gfCNCPoint1[10884] = {X 272.2327, Y 98.0000, Z -1.3333, A 0.000, B 0.000, C 0.000 }
gfCNCPoint1[10885] = {X 272.2329, Y 97.0232, Z -1.3333, A 0.000, B 0.000, C 0.000 }
gfCNCPoint1[10886] = {X 272.3321, Y 96.1797, Z -1.3333, A 0.000, B 0.000, C 0.000 }
gfCNCPoint1[10887] = {X 272.6072, Y 95.3761, Z -1.3333, A 0.000, B 0.000, C 0.000 }
gfCNCPoint1[10888] = {X 273.0457, Y 94.6486, Z -1.3333, A 0.000, B 0.000, C 0.000 }
gfCNCPoint1[10889] = {X 273.6280, Y 94.0302, Z -1.3333, A 0.000, B 0.000, C 0.000 }
gfCNCPoint1[10890] = {X 274.3277, Y 93.5487, Z -1.3333, A 0.000, B 0.000, C 0.000 }
gfCNCPoint1[10891] = {X 275.1133, Y 93.2258, Z -1.3333, A 0.000, B 0.000, C 0.000 }
gfCNCPoint1[10892] = {X 275.9494, Y 93.0760, Z -1.3333, A 0.000, B 0.000, C 0.000 }
gfCNCPoint1[10893] = {X 275.9494, Y 85.3767, Z -1.3333, A 0.000, B 0.000, C 0.000 }
gfCNCPoint1[10894] = {X 262.6059, Y 80.1460, Z -1.3333, A 0.000, B 0.000, C 0.000 }
gfCNCPoint1[10895] = {X 262.1034, Y 80.4620, Z -1.3333, A 0.000, B 0.000, C 0.000 }
gfCNCPoint1[10896] = {X 237.4742, Y 96.4149, Z -1.3333, A 0.000, B 0.000, C 0.000 }
gfCNCPoint1[10897] = {X 237.4798, Y 97.0659, Z -1.3333, A 0.000, B 0.000, C 0.000 }
gfCNCPoint1[10898] = {X 237.4798, Y 98.0000, Z -1.3333, A 0.000, B 0.000, C 0.000 }
gfCNCPoint1[10899] = {X 237.3795, Y 98.8901, Z -1.3333, A 0.000, B 0.000, C 0.000 }
gfCNCPoint1[10900] = {X 237.0837, Y 99.7355, Z -1.3333, A 0.000, B 0.000, C 0.000 }
gfCNCPoint1[10901] = {X 236.6071, Y 100.4940, Z -1.3333, A 0.000, B 0.000, C 0.000 }
gfCNCPoint1[10902] = {X 235.9737, Y 101.1273, Z -1.3333, A 0.000, B 0.000, C 0.000 }
gfCNCPoint1[10903] = {X 235.2153, Y 101.6039, Z -1.3333, A 0.000, B 0.000, C 0.000 }
gfCNCPoint1[10904] = {X 234.3699, Y 101.8997, Z -1.3333, A 0.000, B 0.000, C 0.000 }
gfCNCPoint1[10905] = {X 233.4798, Y 102.0000, Z -1.3333, A 0.000, B 0.000, C 0.000 }
gfCNCPoint1[10906] = {X 214.1790, Y 102.0000, Z -1.3333, A 0.000, B 0.000, C 0.000 }
gfCNCPoint1[10907] = {X 213.7859, Y 101.9806, Z -1.3333, A 0.000, B 0.000, C 0.000 }
gfCNCPoint1[10908] = {X 213.3966, Y 101.9227, Z -1.3333, A 0.000, B 0.000, C 0.000 }
gfCNCPoint1[10909] = {X 213.0072, Y 101.9806, Z -1.3333, A 0.000, B 0.000, C 0.000 }
gfCNCPoint1[10910] = {X 212.6141, Y 102.0000, Z -1.3333, A 0.000, B 0.000, C 0.000 }
gfCNCPoint1[10911] = {X 194.9870, Y 102.0000, Z -1.3333, A 0.000, B 0.000, C 0.000 }
gfCNCPoint1[10912] = {X 194.0969, Y 101.8997, Z -1.3333, A 0.000, B 0.000, C 0.000 }
gfCNCPoint1[10913] = {X 193.2514, Y 101.6039, Z -1.3333, A 0.000, B 0.000, C 0.000 }
gfCNCPoint1[10914] = {X 192.4930, Y 101.1273, Z -1.3333, A 0.000, B 0.000, C 0.000 }
gfCNCPoint1[10915] = {X 191.8596, Y 100.4940, Z -1.3333, A 0.000, B 0.000, C 0.000 }
gfCNCPoint1[10916] = {X 191.3831, Y 99.7355, Z -1.3333, A 0.000, B 0.000, C 0.000 }
gfCNCPoint1[10917] = {X 191.0872, Y 98.8901, Z -1.3333, A 0.000, B 0.000, C 0.000 }
gfCNCPoint1[10918] = {X 190.9870, Y 98.0000, Z -1.3333, A 0.000, B 0.000, C 0.000 }
gfCNCPoint1[10919] = {X 190.9870, Y 97.0659, Z -1.3333, A 0.000, B 0.000, C 0.000 }
gfCNCPoint1[10920] = {X 191.0804, Y 96.2066, Z -1.3333, A 0.000, B 0.000, C 0.000 }
gfCNCPoint1[10921] = {X 191.3562, Y 95.3874, Z -1.3333, A 0.000, B 0.000, C 0.000 }
gfCNCPoint1[10922] = {X 191.8015, Y 94.6466, Z -1.3333, A 0.000, B 0.000, C 0.000 }
gfCNCPoint1[10923] = {X 191.8852, Y 94.5402, Z -1.3333, A 0.000, B 0.000, C 0.000 }
gfCNCPoint1[10924] = {X 191.9725, Y 94.4367, Z -1.3333, A 0.000, B 0.000, C 0.000 }
gfCNCPoint1[10925] = {X 192.0154, Y 94.3938, Z -1.3333, A 0.000, B 0.000, C 0.000 }
gfCNCPoint1[10926] = {X 188.7055, Y 90.7802, Z -1.3333, A 0.000, B 0.000, C 0.000 }
gfCNCPoint1[10927] = {X 149.9476, Y 90.7802, Z -1.3333, A 0.000, B 0.000, C 0.000 }
gfCNCPoint1[10928] = {X 146.7183, Y 94.3579, Z -1.3333, A 0.000, B 0.000, C 0.000 }
gfCNCPoint1[10929] = {X 147.1679, Y 94.9493, Z -1.3333, A 0.000, B 0.000, C 0.000 }
gfCNCPoint1[10930] = {X 147.5014, Y 95.6130, Z -1.3333, A 0.000, B 0.000, C 0.000 }
gfCNCPoint1[10931] = {X 147.7075, Y 96.3267, Z -1.3333, A 0.000, B 0.000, C 0.000 }
gfCNCPoint1[10932] = {X 147.7791, Y 97.0661, Z -1.3333, A 0.000, B 0.000, C 0.000 }
gfCNCPoint1[10933] = {X 147.7791, Y 98.0000, Z -1.3333, A 0.000, B 0.000, C 0.000 }
gfCNCPoint1[10934] = {X 147.6788, Y 98.8901, Z -1.3333, A 0.000, B 0.000, C 0.000 }
gfCNCPoint1[10935] = {X 147.3830, Y 99.7355, Z -1.3333, A 0.000, B 0.000, C 0.000 }
gfCNCPoint1[10936] = {X 146.9064, Y 100.4940, Z -1.3333, A 0.000, B 0.000, C 0.000 }
gfCNCPoint1[10937] = {X 146.2731, Y 101.1273, Z -1.3333, A 0.000, B 0.000, C 0.000 }
gfCNCPoint1[10938] = {X 145.5146, Y 101.6039, Z -1.3333, A 0.000, B 0.000, C 0.000 }
gfCNCPoint1[10939] = {X 144.6692, Y 101.8997, Z -1.3333, A 0.000, B 0.000, C 0.000 }
gfCNCPoint1[10940] = {X 143.7791, Y 102.0000, Z -1.3333, A 0.000, B 0.000, C 0.000 }
gfCNCPoint1[10941] = {X 125.0000, Y 102.0000, Z -1.3333, A 0.000, B 0.000, C 0.000 }
gfCNCPoint1[10942] = {X 124.1099, Y 101.8997, Z -1.3333, A 0.000, B 0.000, C 0.000 }
gfCNCPoint1[10943] = {X 123.2645, Y 101.6039, Z -1.3333, A 0.000, B 0.000, C 0.000 }
gfCNCPoint1[10944] = {X 122.5060, Y 101.1273, Z -1.3333, A 0.000, B 0.000, C 0.000 }
gfCNCPoint1[10945] = {X 121.8727, Y 100.4940, Z -1.3333, A 0.000, B 0.000, C 0.000 }
gfCNCPoint1[10946] = {X 121.3961, Y 99.7355, Z -1.3333, A 0.000, B 0.000, C 0.000 }
gfCNCPoint1[10947] = {X 121.1003, Y 98.8901, Z -1.3333, A 0.000, B 0.000, C 0.000 }
gfCNCPoint1[10948] = {X 121.0000, Y 98.0000, Z -1.3333, A 0.000, B 0.000, C 0.000 }
gfCNCPoint1[10949] = {X 121.0000, Y 97.0659, Z -1.3333, A 0.000, B 0.000, C 0.000 }
gfCNCPoint1[10950] = {X 121.0981, Y 96.1853, Z -1.3333, A 0.000, B 0.000, C 0.000 }
gfCNCPoint1[10951] = {X 121.3877, Y 95.3479, Z -1.3333, A 0.000, B 0.000, C 0.000 }
gfCNCPoint1[10952] = {X 121.8546, Y 94.5948, Z -1.3333, A 0.000, B 0.000, C 0.000 }
gfCNCPoint1[10953] = {X 122.4758, Y 93.9629, Z -1.3333, A 0.000, B 0.000, C 0.000 }
gfCNCPoint1[10954] = {X 123.2209, Y 93.4834, Z -1.3333, A 0.000, B 0.000, C 0.000 }
gfCNCPoint1[10955] = {X 124.0533, Y 93.1796, Z -1.3333, A 0.000, B 0.000, C 0.000 }
gfCNCPoint1[10956] = {X 124.9321, Y 93.0665, Z -1.3333, A 0.000, B 0.000, C 0.000 }
gfCNCPoint1[10957] = {X 124.9750, Y 93.0393, Z -1.3333, A 0.000, B 0.000, C 0.000 }
gfCNCPoint1[10958] = {X 125.4940, Y 92.9623, Z -1.3333, A 0.000, B 0.000, C 0.000 }
gfCNCPoint1[10959] = {X 126.3825, Y 92.8105, Z -1.3333, A 0.000, B 0.000, C 0.000 }
gfCNCPoint1[10960] = {X 127.2582, Y 92.5973, Z -1.3333, A 0.000, B 0.000, C 0.000 }
gfCNCPoint1[10961] = {X 128.5219, Y 91.4099, Z -1.3333, A 0.000, B 0.000, C 0.000 }
gfCNCPoint1[10962] = {X 129.7180, Y 90.1544, Z -1.3333, A 0.000, B 0.000, C 0.000 }
gfCNCPoint1[10963] = {X 133.8038, Y 85.6598, Z -1.3333, A 0.000, B 0.000, C 0.000 }
gfCNCPoint1[10964] = {X 140.9145, Y 77.8539, Z -1.3333, A 0.000, B 0.000, C 0.000 }
gfCNCPoint1[10965] = {X 137.8983, Y 75.1063, Z -1.3333, A 0.000, B 0.000, C 0.000 }
gfCNCPoint1[10966] = {X 137.8983, Y 75.1063, Z 1.6667, A 0.000, B 0.000, C 0.000 }
gfCNCPoint1[10967] = {X 137.8983, Y 75.1063, Z 11.0000, A 0.000, B 0.000, C 0.000 }
gfCNCPoint1[10968] = {X 167.3809, Y 20.2812, Z 11.0000, A 0.000, B 0.000, C 0.000 }
gfCNCPoint1[10969] = {X 167.3809, Y 20.2812, Z 1.6667, A 0.000, B 0.000, C 0.000 }
gfCNCPoint1[10970] = {X 167.3809, Y 20.2812, Z -1.3333, A 0.000, B 0.000, C 0.000 }
gfCNCPoint1[10971] = {X 171.1581, Y 18.7388, Z -1.3333, A 0.000, B 0.000, C 0.000 }
gfCNCPoint1[10972] = {X 169.8405, Y 15.5121, Z -1.3333, A 0.000, B 0.000, C 0.000 }
gfCNCPoint1[10973] = {X 169.5912, Y 14.6607, Z -1.3333, A 0.000, B 0.000, C 0.000 }
gfCNCPoint1[10974] = {X 169.5212, Y 13.7764, Z -1.3333, A 0.000, B 0.000, C 0.000 }
gfCNCPoint1[10975] = {X 169.6332, Y 12.8964, Z -1.3333, A 0.000, B 0.000, C 0.000 }
gfCNCPoint1[10976] = {X 169.9226, Y 12.0578, Z -1.3333, A 0.000, B 0.000, C 0.000 }
gfCNCPoint1[10977] = {X 170.3773, Y 11.2960, Z -1.3333, A 0.000, B 0.000, C 0.000 }
gfCNCPoint1[10978] = {X 170.9779, Y 10.6432, Z -1.3333, A 0.000, B 0.000, C 0.000 }
gfCNCPoint1[10979] = {X 171.6992, Y 10.1268, Z -1.3333, A 0.000, B 0.000, C 0.000 }
gfCNCPoint1[10980] = {X 172.3295, Y 9.7674, Z -1.3333, A 0.000, B 0.000, C 0.000 }
gfCNCPoint1[10981] = {X 173.2114, Y 9.3960, Z -1.3333, A 0.000, B 0.000, C 0.000 }
gfCNCPoint1[10982] = {X 174.1534, Y 9.2278, Z -1.3333, A 0.000, B 0.000, C 0.000 }
gfCNCPoint1[10983] = {X 175.1093, Y 9.2711, Z -1.3333, A 0.000, B 0.000, C 0.000 }
gfCNCPoint1[10984] = {X 176.0323, Y 9.5238, Z -1.3333, A 0.000, B 0.000, C 0.000 }
gfCNCPoint1[10985] = {X 178.2250, Y 8.6014, Z -1.3333, A 0.000, B 0.000, C 0.000 }
gfCNCPoint1[10986] = {X 180.4990, Y 7.9029, Z -1.3333, A 0.000, B 0.000, C 0.000 }
gfCNCPoint1[10987] = {X 182.8314, Y 7.4353, Z -1.3333, A 0.000, B 0.000, C 0.000 }
gfCNCPoint1[10988] = {X 185.1988, Y 7.2031, Z -1.3333, A 0.000, B 0.000, C 0.000 }
gfCNCPoint1[10989] = {X 187.5777, Y 7.2088, Z -1.3333, A 0.000, B 0.000, C 0.000 }
gfCNCPoint1[10990] = {X 189.9440, Y 7.4523, Z -1.3333, A 0.000, B 0.000, C 0.000 }
gfCNCPoint1[10991] = {X 191.7010, Y 7.8143, Z -1.3333, A 0.000, B 0.000, C 0.000 }
gfCNCPoint1[10992] = {X 193.4116, Y 8.3544, Z -1.3333, A 0.000, B 0.000, C 0.000 }
gfCNCPoint1[10993] = {X 195.0579, Y 9.0671, Z -1.3333, A 0.000, B 0.000, C 0.000 }
gfCNCPoint1[10994] = {X 196.6223, Y 9.9449, Z -1.3333, A 0.000, B 0.000, C 0.000 }
gfCNCPoint1[10995] = {X 198.0886, Y 10.9785, Z -1.3333, A 0.000, B 0.000, C 0.000 }
gfCNCPoint1[10996] = {X 199.1482, Y 11.9218, Z -1.3333, A 0.000, B 0.000, C 0.000 }
gfCNCPoint1[10997] = {X 200.0991, Y 12.9747, Z -1.3333, A 0.000, B 0.000, C 0.000 }
gfCNCPoint1[10998] = {X 200.9301, Y 14.1245, Z -1.3333, A 0.000, B 0.000, C 0.000 }
gfCNCPoint1[10999] = {X 201.6314, Y 15.3578, Z -1.3333, A 0.000, B 0.000, C 0.000 }
gfCNCPoint1[11000] = {X 202.1947, Y 16.6598, Z -1.3333, A 0.000, B 0.000, C 0.000 }
gfCNCPoint1[11001] = {X 202.6689, Y 18.3162, Z -1.3333, A 0.000, B 0.000, C 0.000 }
gfCNCPoint1[11002] = {X 202.9504, Y 20.0160, Z -1.3333, A 0.000, B 0.000, C 0.000 }
gfCNCPoint1[11003] = {X 203.0354, Y 21.7368, Z -1.3333, A 0.000, B 0.000, C 0.000 }
gfCNCPoint1[11004] = {X 202.9228, Y 23.4560, Z -1.3333, A 0.000, B 0.000, C 0.000 }
gfCNCPoint1[11005] = {X 202.6141, Y 25.1511, Z -1.3333, A 0.000, B 0.000, C 0.000 }
gfCNCPoint1[11006] = {X 202.1724, Y 26.5972, Z -1.3333, A 0.000, B 0.000, C 0.000 }
gfCNCPoint1[11007] = {X 201.5477, Y 27.9741, Z -1.3333, A 0.000, B 0.000, C 0.000 }
gfCNCPoint1[11008] = {X 200.7505, Y 29.2589, Z -1.3333, A 0.000, B 0.000, C 0.000 }
gfCNCPoint1[11009] = {X 199.7941, Y 30.4301, Z -1.3333, A 0.000, B 0.000, C 0.000 }
gfCNCPoint1[11010] = {X 198.6946, Y 31.4680, Z -1.3333, A 0.000, B 0.000, C 0.000 }
gfCNCPoint1[11011] = {X 199.4963, Y 31.8092, Z -1.3333, A 0.000, B 0.000, C 0.000 }
gfCNCPoint1[11012] = {X 200.2132, Y 32.3043, Z -1.3333, A 0.000, B 0.000, C 0.000 }
gfCNCPoint1[11013] = {X 200.8162, Y 32.9331, Z -1.3333, A 0.000, B 0.000, C 0.000 }
gfCNCPoint1[11014] = {X 201.2808, Y 33.6702, Z -1.3333, A 0.000, B 0.000, C 0.000 }
gfCNCPoint1[11015] = {X 204.3222, Y 39.9530, Z -1.3333, A 0.000, B 0.000, C 0.000 }
gfCNCPoint1[11016] = {X 204.6427, Y 40.8622, Z -1.3333, A 0.000, B 0.000, C 0.000 }
gfCNCPoint1[11017] = {X 204.7537, Y 41.8197, Z -1.3333, A 0.000, B 0.000, C 0.000 }
gfCNCPoint1[11018] = {X 204.6496, Y 42.7781, Z -1.3333, A 0.000, B 0.000, C 0.000 }
gfCNCPoint1[11019] = {X 204.3355, Y 43.6895, Z -1.3333, A 0.000, B 0.000, C 0.000 }
gfCNCPoint1[11020] = {X 203.8272, Y 44.5085, Z -1.3333, A 0.000, B 0.000, C 0.000 }
gfCNCPoint1[11021] = {X 203.1499, Y 45.1945, Z -1.3333, A 0.000, B 0.000, C 0.000 }
gfCNCPoint1[11022] = {X 202.6134, Y 45.6282, Z -1.3333, A 0.000, B 0.000, C 0.000 }
gfCNCPoint1[11023] = {X 201.9086, Y 46.0913, Z -1.3333, A 0.000, B 0.000, C 0.000 }
gfCNCPoint1[11024] = {X 201.1276, Y 46.4092, Z -1.3333, A 0.000, B 0.000, C 0.000 }
gfCNCPoint1[11025] = {X 200.2998, Y 46.5700, Z -1.3333, A 0.000, B 0.000, C 0.000 }
gfCNCPoint1[11026] = {X 199.4565, Y 46.5675, Z -1.3333, A 0.000, B 0.000, C 0.000 }
gfCNCPoint1[11027] = {X 198.6296, Y 46.4019, Z -1.3333, A 0.000, B 0.000, C 0.000 }
gfCNCPoint1[11028] = {X 196.9601, Y 47.2916, Z -1.3333, A 0.000, B 0.000, C 0.000 }
gfCNCPoint1[11029] = {X 195.2345, Y 48.0667, Z -1.3333, A 0.000, B 0.000, C 0.000 }
gfCNCPoint1[11030] = {X 193.4604, Y 48.7236, Z -1.3333, A 0.000, B 0.000, C 0.000 }
gfCNCPoint1[11031] = {X 192.8983, Y 48.9189, Z -1.3333, A 0.000, B 0.000, C 0.000 }
gfCNCPoint1[11032] = {X 190.6740, Y 49.5120, Z -1.3333, A 0.000, B 0.000, C 0.000 }
gfCNCPoint1[11033] = {X 188.4013, Y 49.8784, Z -1.3333, A 0.000, B 0.000, C 0.000 }
gfCNCPoint1[11034] = {X 186.1033, Y 50.0143, Z -1.3333, A 0.000, B 0.000, C 0.000 }
gfCNCPoint1[11035] = {X 183.8033, Y 49.9183, Z -1.3333, A 0.000, B 0.000, C 0.000 }
gfCNCPoint1[11036] = {X 181.5246, Y 49.5914, Z -1.3333, A 0.000, B 0.000, C 0.000 }
gfCNCPoint1[11037] = {X 179.6381, Y 49.1198, Z -1.3333, A 0.000, B 0.000, C 0.000 }
gfCNCPoint1[11038] = {X 177.8176, Y 48.4364, Z -1.3333, A 0.000, B 0.000, C 0.000 }
gfCNCPoint1[11039] = {X 176.0869, Y 47.5499, Z -1.3333, A 0.000, B 0.000, C 0.000 }
gfCNCPoint1[11040] = {X 174.4685, Y 46.4719, Z -1.3333, A 0.000, B 0.000, C 0.000 }
gfCNCPoint1[11041] = {X 173.2359, Y 45.4315, Z -1.3333, A 0.000, B 0.000, C 0.000 }
gfCNCPoint1[11042] = {X 172.1390, Y 44.2489, Z -1.3333, A 0.000, B 0.000, C 0.000 }
gfCNCPoint1[11043] = {X 171.1942, Y 42.9415, Z -1.3333, A 0.000, B 0.000, C 0.000 }
gfCNCPoint1[11044] = {X 170.4154, Y 41.5290, Z -1.3333, A 0.000, B 0.000, C 0.000 }
gfCNCPoint1[11045] = {X 169.8143, Y 40.0322, Z -1.3333, A 0.000, B 0.000, C 0.000 }
gfCNCPoint1[11046] = {X 169.3998, Y 38.4733, Z -1.3333, A 0.000, B 0.000, C 0.000 }
gfCNCPoint1[11047] = {X 169.1779, Y 36.8757, Z -1.3333, A 0.000, B 0.000, C 0.000 }
gfCNCPoint1[11048] = {X 169.0936, Y 35.0419, Z -1.3333, A 0.000, B 0.000, C 0.000 }
gfCNCPoint1[11049] = {X 169.2395, Y 33.2121, Z -1.3333, A 0.000, B 0.000, C 0.000 }
gfCNCPoint1[11050] = {X 169.6135, Y 31.4149, Z -1.3333, A 0.000, B 0.000, C 0.000 }
gfCNCPoint1[11051] = {X 170.2096, Y 29.6787, Z -1.3333, A 0.000, B 0.000, C 0.000 }
gfCNCPoint1[11052] = {X 170.8487, Y 28.3716, Z -1.3333, A 0.000, B 0.000, C 0.000 }
gfCNCPoint1[11053] = {X 171.6568, Y 27.1616, Z -1.3333, A 0.000, B 0.000, C 0.000 }
gfCNCPoint1[11054] = {X 172.6192, Y 26.0704, Z -1.3333, A 0.000, B 0.000, C 0.000 }
gfCNCPoint1[11055] = {X 173.7188, Y 25.1176, Z -1.3333, A 0.000, B 0.000, C 0.000 }
gfCNCPoint1[11056] = {X 174.9359, Y 24.3203, Z -1.3333, A 0.000, B 0.000, C 0.000 }
gfCNCPoint1[11057] = {X 174.1530, Y 23.9327, Z -1.3333, A 0.000, B 0.000, C 0.000 }
gfCNCPoint1[11058] = {X 173.4640, Y 23.3955, Z -1.3333, A 0.000, B 0.000, C 0.000 }
gfCNCPoint1[11059] = {X 172.8972, Y 22.7307, Z -1.3333, A 0.000, B 0.000, C 0.000 }
gfCNCPoint1[11060] = {X 172.4758, Y 21.9655, Z -1.3333, A 0.000, B 0.000, C 0.000 }
gfCNCPoint1[11061] = {X 171.1581, Y 18.7388, Z -1.3333, A 0.000, B 0.000, C 0.000 }
gfCNCPoint1[11062] = {X 167.4550, Y 20.2510, Z -1.3333, A 0.000, B 0.000, C 0.000 }
gfCNCPoint1[11063] = {X 171.2322, Y 18.7085, Z -1.3333, A 0.000, B 0.000, C 0.000 }
gfCNCPoint1[11064] = {X 169.9145, Y 15.4818, Z -1.3333, A 0.000, B 0.000, C 0.000 }
gfCNCPoint1[11065] = {X 169.6699, Y 14.6462, Z -1.3333, A 0.000, B 0.000, C 0.000 }
gfCNCPoint1[11066] = {X 169.6011, Y 13.7783, Z -1.3333, A 0.000, B 0.000, C 0.000 }
gfCNCPoint1[11067] = {X 169.7111, Y 12.9146, Z -1.3333, A 0.000, B 0.000, C 0.000 }
gfCNCPoint1[11068] = {X 169.9952, Y 12.0915, Z -1.3333, A 0.000, B 0.000, C 0.000 }
gfCNCPoint1[11069] = {X 170.4414, Y 11.3439, Z -1.3333, A 0.000, B 0.000, C 0.000 }
gfCNCPoint1[11070] = {X 171.0309, Y 10.7031, Z -1.3333, A 0.000, B 0.000, C 0.000 }
gfCNCPoint1[11071] = {X 171.7389, Y 10.1963, Z -1.3333, A 0.000, B 0.000, C 0.000 }
gfCNCPoint1[11072] = {X 172.3689, Y 9.8371, Z -1.3333, A 0.000, B 0.000, C 0.000 }
gfCNCPoint1[11073] = {X 173.2427, Y 9.4701, Z -1.3333, A 0.000, B 0.000, C 0.000 }
gfCNCPoint1[11074] = {X 174.1763, Y 9.3065, Z -1.3333, A 0.000, B 0.000, C 0.000 }
gfCNCPoint1[11075] = {X 175.1229, Y 9.3543, Z -1.3333, A 0.000, B 0.000, C 0.000 }
gfCNCPoint1[11076] = {X 176.0352, Y 9.6112, Z -1.3333, A 0.000, B 0.000, C 0.000 }
gfCNCPoint1[11077] = {X 178.2247, Y 8.6867, Z -1.3333, A 0.000, B 0.000, C 0.000 }
gfCNCPoint1[11078] = {X 180.4958, Y 7.9863, Z -1.3333, A 0.000, B 0.000, C 0.000 }
gfCNCPoint1[11079] = {X 182.8257, Y 7.5170, Z -1.3333, A 0.000, B 0.000, C 0.000 }
gfCNCPoint1[11080] = {X 185.1909, Y 7.2836, Z -1.3333, A 0.000, B 0.000, C 0.000 }
gfCNCPoint1[11081] = {X 187.5676, Y 7.2884, Z -1.3333, A 0.000, B 0.000, C 0.000 }
gfCNCPoint1[11082] = {X 189.9318, Y 7.5314, Z -1.3333, A 0.000, B 0.000, C 0.000 }
gfCNCPoint1[11083] = {X 191.6808, Y 7.8917, Z -1.3333, A 0.000, B 0.000, C 0.000 }
gfCNCPoint1[11084] = {X 193.3836, Y 8.4294, Z -1.3333, A 0.000, B 0.000, C 0.000 }
gfCNCPoint1[11085] = {X 195.0223, Y 9.1388, Z -1.3333, A 0.000, B 0.000, C 0.000 }
gfCNCPoint1[11086] = {X 196.5797, Y 10.0126, Z -1.3333, A 0.000, B 0.000, C 0.000 }
gfCNCPoint1[11087] = {X 198.0392, Y 11.0414, Z -1.3333, A 0.000, B 0.000, C 0.000 }
gfCNCPoint1[11088] = {X 199.3390, Y 12.2308, Z -1.3333, A 0.000, B 0.000, C 0.000 }
gfCNCPoint1[11089] = {X 200.4656, Y 13.5854, Z -1.3333, A 0.000, B 0.000, C 0.000 }
gfCNCPoint1[11090] = {X 201.3982, Y 15.0802, Z -1.3333, A 0.000, B 0.000, C 0.000 }
gfCNCPoint1[11091] = {X 202.1196, Y 16.6876, Z -1.3333, A 0.000, B 0.000, C 0.000 }
gfCNCPoint1[11092] = {X 202.5911, Y 18.3349, Z -1.3333, A 0.000, B 0.000, C 0.000 }
gfCNCPoint1[11093] = {X 202.8709, Y 20.0254, Z -1.3333, A 0.000, B 0.000, C 0.000 }
gfCNCPoint1[11094] = {X 202.9554, Y 21.7368, Z -1.3333, A 0.000, B 0.000, C 0.000 }
gfCNCPoint1[11095] = {X 202.8433, Y 23.4467, Z -1.3333, A 0.000, B 0.000, C 0.000 }
gfCNCPoint1[11096] = {X 202.5363, Y 25.1324, Z -1.3333, A 0.000, B 0.000, C 0.000 }
gfCNCPoint1[11097] = {X 202.0869, Y 26.5970, Z -1.3333, A 0.000, B 0.000, C 0.000 }
gfCNCPoint1[11098] = {X 201.4485, Y 27.9897, Z -1.3333, A 0.000, B 0.000, C 0.000 }
gfCNCPoint1[11099] = {X 200.6324, Y 29.2861, Z -1.3333, A 0.000, B 0.000, C 0.000 }
gfCNCPoint1[11100] = {X 199.6526, Y 30.4638, Z -1.3333, A 0.000, B 0.000, C 0.000 }
gfCNCPoint1[11101] = {X 198.5263, Y 31.5023, Z -1.3333, A 0.000, B 0.000, C 0.000 }
gfCNCPoint1[11102] = {X 199.3580, Y 31.8261, Z -1.3333, A 0.000, B 0.000, C 0.000 }
gfCNCPoint1[11103] = {X 200.1036, Y 32.3169, Z -1.3333, A 0.000, B 0.000, C 0.000 }
gfCNCPoint1[11104] = {X 200.7299, Y 32.9528, Z -1.3333, A 0.000, B 0.000, C 0.000 }
gfCNCPoint1[11105] = {X 201.2091, Y 33.7058, Z -1.3333, A 0.000, B 0.000, C 0.000 }
gfCNCPoint1[11106] = {X 204.2502, Y 39.9879, Z -1.3333, A 0.000, B 0.000, C 0.000 }
gfCNCPoint1[11107] = {X 204.5648, Y 40.8802, Z -1.3333, A 0.000, B 0.000, C 0.000 }
gfCNCPoint1[11108] = {X 204.6737, Y 41.8200, Z -1.3333, A 0.000, B 0.000, C 0.000 }
gfCNCPoint1[11109] = {X 204.5715, Y 42.7606, Z -1.3333, A 0.000, B 0.000, C 0.000 }
gfCNCPoint1[11110] = {X 204.2633, Y 43.6551, Z -1.3333, A 0.000, B 0.000, C 0.000 }
gfCNCPoint1[11111] = {X 203.7643, Y 44.4590, Z -1.3333, A 0.000, B 0.000, C 0.000 }
gfCNCPoint1[11112] = {X 203.0996, Y 45.1323, Z -1.3333, A 0.000, B 0.000, C 0.000 }
gfCNCPoint1[11113] = {X 202.5632, Y 45.5659, Z -1.3333, A 0.000, B 0.000, C 0.000 }
gfCNCPoint1[11114] = {X 201.8653, Y 46.0237, Z -1.3333, A 0.000, B 0.000, C 0.000 }
gfCNCPoint1[11115] = {X 201.0915, Y 46.3364, Z -1.3333, A 0.000, B 0.000, C 0.000 }
gfCNCPoint1[11116] = {X 200.2715, Y 46.4922, Z -1.3333, A 0.000, B 0.000, C 0.000 }
gfCNCPoint1[11117] = {X 199.4370, Y 46.4850, Z -1.3333, A 0.000, B 0.000, C 0.000 }
gfCNCPoint1[11118] = {X 198.6198, Y 46.3151, Z -1.3333, A 0.000, B 0.000, C 0.000 }
gfCNCPoint1[11119] = {X 196.9456, Y 47.2096, Z -1.3333, A 0.000, B 0.000, C 0.000 }
gfCNCPoint1[11120] = {X 195.2146, Y 47.9884, Z -1.3333, A 0.000, B 0.000, C 0.000 }
gfCNCPoint1[11121] = {X 193.4347, Y 48.6478, Z -1.3333, A 0.000, B 0.000, C 0.000 }
gfCNCPoint1[11122] = {X 192.8729, Y 48.8430, Z -1.3333, A 0.000, B 0.000, C 0.000 }
gfCNCPoint1[11123] = {X 190.6565, Y 49.4340, Z -1.3333, A 0.000, B 0.000, C 0.000 }
gfCNCPoint1[11124] = {X 188.3919, Y 49.7990, Z -1.3333, A 0.000, B 0.000, C 0.000 }
gfCNCPoint1[11125] = {X 186.1021, Y 49.9343, Z -1.3333, A 0.000, B 0.000, C 0.000 }
gfCNCPoint1[11126] = {X 183.8103, Y 49.8386, Z -1.3333, A 0.000, B 0.000, C 0.000 }
gfCNCPoint1[11127] = {X 181.5397, Y 49.5128, Z -1.3333, A 0.000, B 0.000, C 0.000 }
gfCNCPoint1[11128] = {X 179.6620, Y 49.0435, Z -1.3333, A 0.000, B 0.000, C 0.000 }
gfCNCPoint1[11129] = {X 177.8500, Y 48.3632, Z -1.3333, A 0.000, B 0.000, C 0.000 }
gfCNCPoint1[11130] = {X 176.1274, Y 47.4809, Z -1.3333, A 0.000, B 0.000, C 0.000 }
gfCNCPoint1[11131] = {X 174.5165, Y 46.4079, Z -1.3333, A 0.000, B 0.000, C 0.000 }
gfCNCPoint1[11132] = {X 173.2911, Y 45.3737, Z -1.3333, A 0.000, B 0.000, C 0.000 }
gfCNCPoint1[11133] = {X 172.2008, Y 44.1980, Z -1.3333, A 0.000, B 0.000, C 0.000 }
gfCNCPoint1[11134] = {X 171.2616, Y 42.8984, Z -1.3333, A 0.000, B 0.000, C 0.000 }
gfCNCPoint1[11135] = {X 170.4874, Y 41.4941, Z -1.3333, A 0.000, B 0.000, C 0.000 }
gfCNCPoint1[11136] = {X 169.8900, Y 40.0061, Z -1.3333, A 0.000, B 0.000, C 0.000 }
gfCNCPoint1[11137] = {X 169.4780, Y 38.4565, Z -1.3333, A 0.000, B 0.000, C 0.000 }
gfCNCPoint1[11138] = {X 169.2576, Y 36.8682, Z -1.3333, A 0.000, B 0.000, C 0.000 }
gfCNCPoint1[11139] = {X 169.1736, Y 35.0442, Z -1.3333, A 0.000, B 0.000, C 0.000 }
gfCNCPoint1[11140] = {X 169.3187, Y 33.2239, Z -1.3333, A 0.000, B 0.000, C 0.000 }
gfCNCPoint1[11141] = {X 169.6906, Y 31.4362, Z -1.3333, A 0.000, B 0.000, C 0.000 }
gfCNCPoint1[11142] = {X 170.2836, Y 29.7091, Z -1.3333, A 0.000, B 0.000, C 0.000 }
gfCNCPoint1[11143] = {X 170.9358, Y 28.3808, Z -1.3333, A 0.000, B 0.000, C 0.000 }
gfCNCPoint1[11144] = {X 171.7637, Y 27.1542, Z -1.3333, A 0.000, B 0.000, C 0.000 }
gfCNCPoint1[11145] = {X 172.7517, Y 26.0525, Z -1.3333, A 0.000, B 0.000, C 0.000 }
gfCNCPoint1[11146] = {X 173.8812, Y 25.0964, Z -1.3333, A 0.000, B 0.000, C 0.000 }
gfCNCPoint1[11147] = {X 175.1309, Y 24.3039, Z -1.3333, A 0.000, B 0.000, C 0.000 }
gfCNCPoint1[11148] = {X 174.3091, Y 23.9338, Z -1.3333, A 0.000, B 0.000, C 0.000 }
gfCNCPoint1[11149] = {X 173.5841, Y 23.3984, Z -1.3333, A 0.000, B 0.000, C 0.000 }
gfCNCPoint1[11150] = {X 172.9886, Y 22.7218, Z -1.3333, A 0.000, B 0.000, C 0.000 }
gfCNCPoint1[11151] = {X 172.5496, Y 21.9347, Z -1.3333, A 0.000, B 0.000, C 0.000 }
gfCNCPoint1[11152] = {X 171.2322, Y 18.7085, Z -1.3333, A 0.000, B 0.000, C 0.000 }
gfCNCPoint1[11153] = {X 167.5291, Y 20.2207, Z -1.3333, A 0.000, B 0.000, C 0.000 }
gfCNCPoint1[11154] = {X 171.3062, Y 18.6783, Z -1.3333, A 0.000, B 0.000, C 0.000 }
gfCNCPoint1[11155] = {X 169.9886, Y 15.4516, Z -1.3333, A 0.000, B 0.000, C 0.000 }
gfCNCPoint1[11156] = {X 169.7252, Y 14.4911, Z -1.3333, A 0.000, B 0.000, C 0.000 }
gfCNCPoint1[11157] = {X 169.6977, Y 13.4955, Z -1.3333, A 0.000, B 0.000, C 0.000 }
gfCNCPoint1[11158] = {X 169.9076, Y 12.5218, Z -1.3333, A 0.000, B 0.000, C 0.000 }
gfCNCPoint1[11159] = {X 170.3429, Y 11.6260, Z -1.3333, A 0.000, B 0.000, C 0.000 }
gfCNCPoint1[11160] = {X 170.9787, Y 10.8594, Z -1.3333, A 0.000, B 0.000, C 0.000 }
gfCNCPoint1[11161] = {X 171.7785, Y 10.2658, Z -1.3333, A 0.000, B 0.000, C 0.000 }
gfCNCPoint1[11162] = {X 172.4082, Y 9.9068, Z -1.3333, A 0.000, B 0.000, C 0.000 }
gfCNCPoint1[11163] = {X 173.2740, Y 9.5443, Z -1.3333, A 0.000, B 0.000, C 0.000 }
gfCNCPoint1[11164] = {X 174.1991, Y 9.3853, Z -1.3333, A 0.000, B 0.000, C 0.000 }
gfCNCPoint1[11165] = {X 175.1362, Y 9.4376, Z -1.3333, A 0.000, B 0.000, C 0.000 }
gfCNCPoint1[11166] = {X 176.0378, Y 9.6988, Z -1.3333, A 0.000, B 0.000, C 0.000 }
gfCNCPoint1[11167] = {X 178.2241, Y 8.7721, Z -1.3333, A 0.000, B 0.000, C 0.000 }
gfCNCPoint1[11168] = {X 180.4925, Y 8.0697, Z -1.3333, A 0.000, B 0.000, C 0.000 }
gfCNCPoint1[11169] = {X 182.8199, Y 7.5988, Z -1.3333, A 0.000, B 0.000, C 0.000 }
gfCNCPoint1[11170] = {X 185.1829, Y 7.3641, Z -1.3333, A 0.000, B 0.000, C 0.000 }
gfCNCPoint1[11171] = {X 187.5575, Y 7.3680, Z -1.3333, A 0.000, B 0.000, C 0.000 }
gfCNCPoint1[11172] = {X 189.9197, Y 7.6105, Z -1.3333, A 0.000, B 0.000, C 0.000 }
gfCNCPoint1[11173] = {X 191.6606, Y 7.9691, Z -1.3333, A 0.000, B 0.000, C 0.000 }
gfCNCPoint1[11174] = {X 193.3556, Y 8.5043, Z -1.3333, A 0.000, B 0.000, C 0.000 }
gfCNCPoint1[11175] = {X 194.9868, Y 9.2105, Z -1.3333, A 0.000, B 0.000, C 0.000 }
gfCNCPoint1[11176] = {X 196.5370, Y 10.0802, Z -1.3333, A 0.000, B 0.000, C 0.000 }
gfCNCPoint1[11177] = {X 197.9898, Y 11.1043, Z -1.3333, A 0.000, B 0.000, C 0.000 }
gfCNCPoint1[11178] = {X 199.2813, Y 12.2862, Z -1.3333, A 0.000, B 0.000, C 0.000 }
gfCNCPoint1[11179] = {X 200.4007, Y 13.6322, Z -1.3333, A 0.000, B 0.000, C 0.000 }
gfCNCPoint1[11180] = {X 201.3274, Y 15.1175, Z -1.3333, A 0.000, B 0.000, C 0.000 }
gfCNCPoint1[11181] = {X 202.0443, Y 16.7146, Z -1.3333, A 0.000, B 0.000, C 0.000 }
gfCNCPoint1[11182] = {X 202.5132, Y 18.3531, Z -1.3333, A 0.000, B 0.000, C 0.000 }
gfCNCPoint1[11183] = {X 202.7914, Y 20.0344, Z -1.3333, A 0.000, B 0.000, C 0.000 }
gfCNCPoint1[11184] = {X 202.8754, Y 21.7366, Z -1.3333, A 0.000, B 0.000, C 0.000 }
gfCNCPoint1[11185] = {X 202.7639, Y 23.4372, Z -1.3333, A 0.000, B 0.000, C 0.000 }
gfCNCPoint1[11186] = {X 202.4585, Y 25.1138, Z -1.3333, A 0.000, B 0.000, C 0.000 }
gfCNCPoint1[11187] = {X 202.0007, Y 26.5985, Z -1.3333, A 0.000, B 0.000, C 0.000 }
gfCNCPoint1[11188] = {X 201.3474, Y 28.0081, Z -1.3333, A 0.000, B 0.000, C 0.000 }
gfCNCPoint1[11189] = {X 200.5105, Y 29.3171, Z -1.3333, A 0.000, B 0.000, C 0.000 }
gfCNCPoint1[11190] = {X 199.5053, Y 30.5017, Z -1.3333, A 0.000, B 0.000, C 0.000 }
gfCNCPoint1[11191] = {X 198.3499, Y 31.5404, Z -1.3333, A 0.000, B 0.000, C 0.000 }
gfCNCPoint1[11192] = {X 199.2138, Y 31.8436, Z -1.3333, A 0.000, B 0.000, C 0.000 }
gfCNCPoint1[11193] = {X 199.9904, Y 32.3284, Z -1.3333, A 0.000, B 0.000, C 0.000 }
gfCNCPoint1[11194] = {X 200.6422, Y 32.9714, Z -1.3333, A 0.000, B 0.000, C 0.000 }
gfCNCPoint1[11195] = {X 201.1375, Y 33.7414, Z -1.3333, A 0.000, B 0.000, C 0.000 }
gfCNCPoint1[11196] = {X 204.1781, Y 40.0227, Z -1.3333, A 0.000, B 0.000, C 0.000 }
gfCNCPoint1[11197] = {X 204.4868, Y 40.8982, Z -1.3333, A 0.000, B 0.000, C 0.000 }
gfCNCPoint1[11198] = {X 204.5937, Y 41.8203, Z -1.3333, A 0.000, B 0.000, C 0.000 }
gfCNCPoint1[11199] = {X 204.4934, Y 42.7431, Z -1.3333, A 0.000, B 0.000, C 0.000 }
gfCNCPoint1[11200] = {X 204.1910, Y 43.6208, Z -1.3333, A 0.000, B 0.000, C 0.000 }
gfCNCPoint1[11201] = {X 203.7015, Y 44.4095, Z -1.3333, A 0.000, B 0.000, C 0.000 }
gfCNCPoint1[11202] = {X 203.0493, Y 45.0700, Z -1.3333, A 0.000, B 0.000, C 0.000 }
gfCNCPoint1[11203] = {X 202.5130, Y 45.5037, Z -1.3333, A 0.000, B 0.000, C 0.000 }
gfCNCPoint1[11204] = {X 201.8220, Y 45.9561, Z -1.3333, A 0.000, B 0.000, C 0.000 }
gfCNCPoint1[11205] = {X 201.0555, Y 46.2636, Z -1.3333, A 0.000, B 0.000, C 0.000 }
gfCNCPoint1[11206] = {X 200.2434, Y 46.4144, Z -1.3333, A 0.000, B 0.000, C 0.000 }
gfCNCPoint1[11207] = {X 199.4176, Y 46.4024, Z -1.3333, A 0.000, B 0.000, C 0.000 }
gfCNCPoint1[11208] = {X 198.6103, Y 46.2282, Z -1.3333, A 0.000, B 0.000, C 0.000 }
gfCNCPoint1[11209] = {X 196.9313, Y 47.1275, Z -1.3333, A 0.000, B 0.000, C 0.000 }
gfCNCPoint1[11210] = {X 195.1948, Y 47.9100, Z -1.3333, A 0.000, B 0.000, C 0.000 }
gfCNCPoint1[11211] = {X 193.4089, Y 48.5721, Z -1.3333, A 0.000, B 0.000, C 0.000 }
gfCNCPoint1[11212] = {X 192.8475, Y 48.7671, Z -1.3333, A 0.000, B 0.000, C 0.000 }
gfCNCPoint1[11213] = {X 190.6391, Y 49.3559, Z -1.3333, A 0.000, B 0.000, C 0.000 }
gfCNCPoint1[11214] = {X 188.3826, Y 49.7195, Z -1.3333, A 0.000, B 0.000, C 0.000 }
gfCNCPoint1[11215] = {X 186.1010, Y 49.8543, Z -1.3333, A 0.000, B 0.000, C 0.000 }
gfCNCPoint1[11216] = {X 183.8173, Y 49.7589, Z -1.3333, A 0.000, B 0.000, C 0.000 }
gfCNCPoint1[11217] = {X 181.5549, Y 49.4343, Z -1.3333, A 0.000, B 0.000, C 0.000 }
gfCNCPoint1[11218] = {X 179.6860, Y 48.9672, Z -1.3333, A 0.000, B 0.000, C 0.000 }
gfCNCPoint1[11219] = {X 177.8824, Y 48.2901, Z -1.3333, A 0.000, B 0.000, C 0.000 }
gfCNCPoint1[11220] = {X 176.1678, Y 47.4118, Z -1.3333, A 0.000, B 0.000, C 0.000 }
gfCNCPoint1[11221] = {X 174.5644, Y 46.3439, Z -1.3333, A 0.000, B 0.000, C 0.000 }
gfCNCPoint1[11222] = {X 173.3464, Y 45.3158, Z -1.3333, A 0.000, B 0.000, C 0.000 }
gfCNCPoint1[11223] = {X 172.2625, Y 44.1471, Z -1.3333, A 0.000, B 0.000, C 0.000 }
gfCNCPoint1[11224] = {X 171.3289, Y 42.8552, Z -1.3333, A 0.000, B 0.000, C 0.000 }
gfCNCPoint1[11225] = {X 170.5595, Y 41.4593, Z -1.3333, A 0.000, B 0.000, C 0.000 }
gfCNCPoint1[11226] = {X 169.9656, Y 39.9801, Z -1.3333, A 0.000, B 0.000, C 0.000 }
gfCNCPoint1[11227] = {X 169.5562, Y 38.4396, Z -1.3333, A 0.000, B 0.000, C 0.000 }
gfCNCPoint1[11228] = {X 169.3373, Y 36.8608, Z -1.3333, A 0.000, B 0.000, C 0.000 }
gfCNCPoint1[11229] = {X 169.2535, Y 35.0464, Z -1.3333, A 0.000, B 0.000, C 0.000 }
gfCNCPoint1[11230] = {X 169.3978, Y 33.2358, Z -1.3333, A 0.000, B 0.000, C 0.000 }
gfCNCPoint1[11231] = {X 169.7677, Y 31.4575, Z -1.3333, A 0.000, B 0.000, C 0.000 }
gfCNCPoint1[11232] = {X 170.3575, Y 29.7396, Z -1.3333, A 0.000, B 0.000, C 0.000 }
gfCNCPoint1[11233] = {X 171.0244, Y 28.3876, Z -1.3333, A 0.000, B 0.000, C 0.000 }
gfCNCPoint1[11234] = {X 171.8745, Y 27.1426, Z -1.3333, A 0.000, B 0.000, C 0.000 }
gfCNCPoint1[11235] = {X 172.8911, Y 26.0294, Z -1.3333, A 0.000, B 0.000, C 0.000 }
gfCNCPoint1[11236] = {X 174.0540, Y 25.0701, Z -1.3333, A 0.000, B 0.000, C 0.000 }
gfCNCPoint1[11237] = {X 175.3400, Y 24.2836, Z -1.3333, A 0.000, B 0.000, C 0.000 }
gfCNCPoint1[11238] = {X 174.4755, Y 23.9356, Z -1.3333, A 0.000, B 0.000, C 0.000 }
gfCNCPoint1[11239] = {X 173.7101, Y 23.4039, Z -1.3333, A 0.000, B 0.000, C 0.000 }
gfCNCPoint1[11240] = {X 173.0822, Y 22.7151, Z -1.3333, A 0.000, B 0.000, C 0.000 }
gfCNCPoint1[11241] = {X 172.6235, Y 21.9039, Z -1.3333, A 0.000, B 0.000, C 0.000 }
gfCNCPoint1[11242] = {X 171.3062, Y 18.6783, Z -1.3333, A 0.000, B 0.000, C 0.000 }
gfCNCPoint1[11243] = {X 167.6031, Y 20.1905, Z -1.3333, A 0.000, B 0.000, C 0.000 }
gfCNCPoint1[11244] = {X 171.3803, Y 18.6480, Z -1.3333, A 0.000, B 0.000, C 0.000 }
gfCNCPoint1[11245] = {X 170.0626, Y 15.4213, Z -1.3333, A 0.000, B 0.000, C 0.000 }
gfCNCPoint1[11246] = {X 169.8043, Y 14.4793, Z -1.3333, A 0.000, B 0.000, C 0.000 }
gfCNCPoint1[11247] = {X 169.7773, Y 13.5028, Z -1.3333, A 0.000, B 0.000, C 0.000 }
gfCNCPoint1[11248] = {X 169.9832, Y 12.5479, Z -1.3333, A 0.000, B 0.000, C 0.000 }
gfCNCPoint1[11249] = {X 170.4102, Y 11.6694, Z -1.3333, A 0.000, B 0.000, C 0.000 }
gfCNCPoint1[11250] = {X 171.0337, Y 10.9174, Z -1.3333, A 0.000, B 0.000, C 0.000 }
gfCNCPoint1[11251] = {X 171.8181, Y 10.3353, Z -1.3333, A 0.000, B 0.000, C 0.000 }
gfCNCPoint1[11252] = {X 172.4475, Y 9.9764, Z -1.3333, A 0.000, B 0.000, C 0.000 }
gfCNCPoint1[11253] = {X 173.3053, Y 9.6186, Z -1.3333, A 0.000, B 0.000, C 0.000 }
gfCNCPoint1[11254] = {X 174.2218, Y 9.4641, Z -1.3333, A 0.000, B 0.000, C 0.000 }
gfCNCPoint1[11255] = {X 175.1494, Y 9.5211, Z -1.3333, A 0.000, B 0.000, C 0.000 }
gfCNCPoint1[11256] = {X 176.0401, Y 9.7866, Z -1.3333, A 0.000, B 0.000, C 0.000 }
gfCNCPoint1[11257] = {X 178.2233, Y 8.8576, Z -1.3333, A 0.000, B 0.000, C 0.000 }
gfCNCPoint1[11258] = {X 180.4889, Y 8.1532, Z -1.3333, A 0.000, B 0.000, C 0.000 }
gfCNCPoint1[11259] = {X 182.8139, Y 7.6806, Z -1.3333, A 0.000, B 0.000, C 0.000 }
gfCNCPoint1[11260] = {X 185.1747, Y 7.4446, Z -1.3333, A 0.000, B 0.000, C 0.000 }
gfCNCPoint1[11261] = {X 187.5473, Y 7.4476, Z -1.3333, A 0.000, B 0.000, C 0.000 }
gfCNCPoint1[11262] = {X 189.9075, Y 7.6895, Z -1.3333, A 0.000, B 0.000, C 0.000 }
gfCNCPoint1[11263] = {X 191.6404, Y 8.0465, Z -1.3333, A 0.000, B 0.000, C 0.000 }
gfCNCPoint1[11264] = {X 193.3276, Y 8.5792, Z -1.3333, A 0.000, B 0.000, C 0.000 }
gfCNCPoint1[11265] = {X 194.9513, Y 9.2822, Z -1.3333, A 0.000, B 0.000, C 0.000 }
gfCNCPoint1[11266] = {X 196.4943, Y 10.1479, Z -1.3333, A 0.000, B 0.000, C 0.000 }
gfCNCPoint1[11267] = {X 197.9404, Y 11.1673, Z -1.3333, A 0.000, B 0.000, C 0.000 }
gfCNCPoint1[11268] = {X 199.2236, Y 12.3417, Z -1.3333, A 0.000, B 0.000, C 0.000 }
gfCNCPoint1[11269] = {X 200.3358, Y 13.6791, Z -1.3333, A 0.000, B 0.000, C 0.000 }
gfCNCPoint1[11270] = {X 201.2566, Y 15.1548, Z -1.3333, A 0.000, B 0.000, C 0.000 }
gfCNCPoint1[11271] = {X 201.9691, Y 16.7417, Z -1.3333, A 0.000, B 0.000, C 0.000 }
gfCNCPoint1[11272] = {X 202.4353, Y 18.3712, Z -1.3333, A 0.000, B 0.000, C 0.000 }
gfCNCPoint1[11273] = {X 202.7119, Y 20.0435, Z -1.3333, A 0.000, B 0.000, C 0.000 }
gfCNCPoint1[11274] = {X 202.7954, Y 21.7364, Z -1.3333, A 0.000, B 0.000, C 0.000 }
gfCNCPoint1[11275] = {X 202.6845, Y 23.4277, Z -1.3333, A 0.000, B 0.000, C 0.000 }
gfCNCPoint1[11276] = {X 202.3807, Y 25.0952, Z -1.3333, A 0.000, B 0.000, C 0.000 }
gfCNCPoint1[11277] = {X 201.9136, Y 26.6019, Z -1.3333, A 0.000, B 0.000, C 0.000 }
gfCNCPoint1[11278] = {X 201.2439, Y 28.0301, Z -1.3333, A 0.000, B 0.000, C 0.000 }
gfCNCPoint1[11279] = {X 200.3842, Y 29.3527, Z -1.3333, A 0.000, B 0.000, C 0.000 }
gfCNCPoint1[11280] = {X 199.3509, Y 30.5446, Z -1.3333, A 0.000, B 0.000, C 0.000 }
gfCNCPoint1[11281] = {X 198.1636, Y 31.5831, Z -1.3333, A 0.000, B 0.000, C 0.000 }
gfCNCPoint1[11282] = {X 199.0619, Y 31.8617, Z -1.3333, A 0.000, B 0.000, C 0.000 }
gfCNCPoint1[11283] = {X 199.8726, Y 32.3385, Z -1.3333, A 0.000, B 0.000, C 0.000 }
gfCNCPoint1[11284] = {X 200.5526, Y 32.9884, Z -1.3333, A 0.000, B 0.000, C 0.000 }
gfCNCPoint1[11285] = {X 201.0657, Y 33.7766, Z -1.3333, A 0.000, B 0.000, C 0.000 }
gfCNCPoint1[11286] = {X 204.1061, Y 40.0576, Z -1.3333, A 0.000, B 0.000, C 0.000 }
gfCNCPoint1[11287] = {X 204.4089, Y 40.9162, Z -1.3333, A 0.000, B 0.000, C 0.000 }
gfCNCPoint1[11288] = {X 204.5137, Y 41.8206, Z -1.3333, A 0.000, B 0.000, C 0.000 }
gfCNCPoint1[11289] = {X 204.4154, Y 42.7257, Z -1.3333, A 0.000, B 0.000, C 0.000 }
gfCNCPoint1[11290] = {X 204.1188, Y 43.5864, Z -1.3333, A 0.000, B 0.000, C 0.000 }
gfCNCPoint1[11291] = {X 203.6387, Y 44.3600, Z -1.3333, A 0.000, B 0.000, C 0.000 }
gfCNCPoint1[11292] = {X 202.9990, Y 45.0078, Z -1.3333, A 0.000, B 0.000, C 0.000 }
gfCNCPoint1[11293] = {X 202.4628, Y 45.4414, Z -1.3333, A 0.000, B 0.000, C 0.000 }
gfCNCPoint1[11294] = {X 201.7787, Y 45.8884, Z -1.3333, A 0.000, B 0.000, C 0.000 }
gfCNCPoint1[11295] = {X 201.0195, Y 46.1907, Z -1.3333, A 0.000, B 0.000, C 0.000 }
gfCNCPoint1[11296] = {X 200.2155, Y 46.3364, Z -1.3333, A 0.000, B 0.000, C 0.000 }
gfCNCPoint1[11297] = {X 199.3985, Y 46.3196, Z -1.3333, A 0.000, B 0.000, C 0.000 }
gfCNCPoint1[11298] = {X 198.6011, Y 46.1410, Z -1.3333, A 0.000, B 0.000, C 0.000 }
gfCNCPoint1[11299] = {X 196.9172, Y 47.0453, Z -1.3333, A 0.000, B 0.000, C 0.000 }
gfCNCPoint1[11300] = {X 195.1752, Y 47.8316, Z -1.3333, A 0.000, B 0.000, C 0.000 }
gfCNCPoint1[11301] = {X 193.3832, Y 48.4963, Z -1.3333, A 0.000, B 0.000, C 0.000 }
gfCNCPoint1[11302] = {X 192.8222, Y 48.6912, Z -1.3333, A 0.000, B 0.000, C 0.000 }
gfCNCPoint1[11303] = {X 190.6216, Y 49.2778, Z -1.3333, A 0.000, B 0.000, C 0.000 }
gfCNCPoint1[11304] = {X 188.3732, Y 49.6401, Z -1.3333, A 0.000, B 0.000, C 0.000 }
gfCNCPoint1[11305] = {X 186.0998, Y 49.7743, Z -1.3333, A 0.000, B 0.000, C 0.000 }
gfCNCPoint1[11306] = {X 183.8244, Y 49.6792, Z -1.3333, A 0.000, B 0.000, C 0.000 }
gfCNCPoint1[11307] = {X 181.5701, Y 49.3557, Z -1.3333, A 0.000, B 0.000, C 0.000 }
gfCNCPoint1[11308] = {X 179.7099, Y 48.8908, Z -1.3333, A 0.000, B 0.000, C 0.000 }
gfCNCPoint1[11309] = {X 177.9148, Y 48.2169, Z -1.3333, A 0.000, B 0.000, C 0.000 }
gfCNCPoint1[11310] = {X 176.2082, Y 47.3428, Z -1.3333, A 0.000, B 0.000, C 0.000 }
gfCNCPoint1[11311] = {X 174.6124, Y 46.2799, Z -1.3333, A 0.000, B 0.000, C 0.000 }
gfCNCPoint1[11312] = {X 173.4016, Y 45.2579, Z -1.3333, A 0.000, B 0.000, C 0.000 }
gfCNCPoint1[11313] = {X 172.3242, Y 44.0962, Z -1.3333, A 0.000, B 0.000, C 0.000 }
gfCNCPoint1[11314] = {X 171.3962, Y 42.8120, Z -1.3333, A 0.000, B 0.000, C 0.000 }
gfCNCPoint1[11315] = {X 170.6315, Y 41.4244, Z -1.3333, A 0.000, B 0.000, C 0.000 }
gfCNCPoint1[11316] = {X 170.0413, Y 39.9541, Z -1.3333, A 0.000, B 0.000, C 0.000 }
gfCNCPoint1[11317] = {X 169.6344, Y 38.4228, Z -1.3333, A 0.000, B 0.000, C 0.000 }
gfCNCPoint1[11318] = {X 169.4169, Y 36.8534, Z -1.3333, A 0.000, B 0.000, C 0.000 }
gfCNCPoint1[11319] = {X 169.3335, Y 35.0486, Z -1.3333, A 0.000, B 0.000, C 0.000 }
gfCNCPoint1[11320] = {X 169.4769, Y 33.2476, Z -1.3333, A 0.000, B 0.000, C 0.000 }
gfCNCPoint1[11321] = {X 169.8448, Y 31.4788, Z -1.3333, A 0.000, B 0.000, C 0.000 }
gfCNCPoint1[11322] = {X 170.4315, Y 29.7700, Z -1.3333, A 0.000, B 0.000, C 0.000 }
gfCNCPoint1[11323] = {X 171.1150, Y 28.3912, Z -1.3333, A 0.000, B 0.000, C 0.000 }
gfCNCPoint1[11324] = {X 171.9906, Y 27.1255, Z -1.3333, A 0.000, B 0.000, C 0.000 }
gfCNCPoint1[11325] = {X 173.0398, Y 25.9995, Z -1.3333, A 0.000, B 0.000, C 0.000 }
gfCNCPoint1[11326] = {X 174.2406, Y 25.0370, Z -1.3333, A 0.000, B 0.000, C 0.000 }
gfCNCPoint1[11327] = {X 175.5679, Y 24.2580, Z -1.3333, A 0.000, B 0.000, C 0.000 }
gfCNCPoint1[11328] = {X 174.6555, Y 23.9383, Z -1.3333, A 0.000, B 0.000, C 0.000 }
gfCNCPoint1[11329] = {X 173.8439, Y 23.4130, Z -1.3333, A 0.000, B 0.000, C 0.000 }
gfCNCPoint1[11330] = {X 173.1788, Y 22.7114, Z -1.3333, A 0.000, B 0.000, C 0.000 }
gfCNCPoint1[11331] = {X 172.6973, Y 21.8731, Z -1.3333, A 0.000, B 0.000, C 0.000 }
gfCNCPoint1[11332] = {X 171.3803, Y 18.6480, Z -1.3333, A 0.000, B 0.000, C 0.000 }
gfCNCPoint1[11333] = {X 167.6770, Y 20.1603, Z -1.3333, A 0.000, B 0.000, C 0.000 }
gfCNCPoint1[11334] = {X 167.6769, Y 20.1601, Z -1.3333, A 0.000, B 0.000, C 0.000 }
gfCNCPoint1[11335] = {X 171.4542, Y 18.6179, Z -1.3333, A 0.000, B 0.000, C 0.000 }
gfCNCPoint1[11336] = {X 170.1367, Y 15.3911, Z -1.3333, A 0.000, B 0.000, C 0.000 }
gfCNCPoint1[11337] = {X 169.8835, Y 14.4675, Z -1.3333, A 0.000, B 0.000, C 0.000 }
gfCNCPoint1[11338] = {X 169.8570, Y 13.5102, Z -1.3333, A 0.000, B 0.000, C 0.000 }
gfCNCPoint1[11339] = {X 170.0588, Y 12.5740, Z -1.3333, A 0.000, B 0.000, C 0.000 }
gfCNCPoint1[11340] = {X 170.4774, Y 11.7127, Z -1.3333, A 0.000, B 0.000, C 0.000 }
gfCNCPoint1[11341] = {X 171.0888, Y 10.9755, Z -1.3333, A 0.000, B 0.000, C 0.000 }
gfCNCPoint1[11342] = {X 171.8578, Y 10.4048, Z -1.3333, A 0.000, B 0.000, C 0.000 }
gfCNCPoint1[11343] = {X 172.4867, Y 10.0462, Z -1.3333, A 0.000, B 0.000, C 0.000 }
gfCNCPoint1[11344] = {X 173.3363, Y 9.6929, Z -1.3333, A 0.000, B 0.000, C 0.000 }
gfCNCPoint1[11345] = {X 174.2443, Y 9.5431, Z -1.3333, A 0.000, B 0.000, C 0.000 }
gfCNCPoint1[11346] = {X 175.1624, Y 9.6048, Z -1.3333, A 0.000, B 0.000, C 0.000 }
gfCNCPoint1[11347] = {X 176.0421, Y 9.8746, Z -1.3333, A 0.000, B 0.000, C 0.000 }
gfCNCPoint1[11348] = {X 178.2221, Y 8.9432, Z -1.3333, A 0.000, B 0.000, C 0.000 }
gfCNCPoint1[11349] = {X 180.4850, Y 8.2368, Z -1.3333, A 0.000, B 0.000, C 0.000 }
gfCNCPoint1[11350] = {X 182.8077, Y 7.7624, Z -1.3333, A 0.000, B 0.000, C 0.000 }
gfCNCPoint1[11351] = {X 185.1664, Y 7.5251, Z -1.3333, A 0.000, B 0.000, C 0.000 }
gfCNCPoint1[11352] = {X 187.5371, Y 7.5272, Z -1.3333, A 0.000, B 0.000, C 0.000 }
gfCNCPoint1[11353] = {X 189.8953, Y 7.7686, Z -1.3333, A 0.000, B 0.000, C 0.000 }
gfCNCPoint1[11354] = {X 191.6202, Y 8.1239, Z -1.3333, A 0.000, B 0.000, C 0.000 }
gfCNCPoint1[11355] = {X 193.2996, Y 8.6542, Z -1.3333, A 0.000, B 0.000, C 0.000 }
gfCNCPoint1[11356] = {X 194.9157, Y 9.3538, Z -1.3333, A 0.000, B 0.000, C 0.000 }
gfCNCPoint1[11357] = {X 196.4516, Y 10.2156, Z -1.3333, A 0.000, B 0.000, C 0.000 }
gfCNCPoint1[11358] = {X 197.8910, Y 11.2302, Z -1.3333, A 0.000, B 0.000, C 0.000 }
gfCNCPoint1[11359] = {X 199.1659, Y 12.3971, Z -1.3333, A 0.000, B 0.000, C 0.000 }
gfCNCPoint1[11360] = {X 200.2710, Y 13.7259, Z -1.3333, A 0.000, B 0.000, C 0.000 }
gfCNCPoint1[11361] = {X 201.1859, Y 15.1921, Z -1.3333, A 0.000, B 0.000, C 0.000 }
gfCNCPoint1[11362] = {X 201.8938, Y 16.7687, Z -1.3333, A 0.000, B 0.000, C 0.000 }
gfCNCPoint1[11363] = {X 202.3574, Y 18.3894, Z -1.3333, A 0.000, B 0.000, C 0.000 }
gfCNCPoint1[11364] = {X 202.6324, Y 20.0525, Z -1.3333, A 0.000, B 0.000, C 0.000 }
gfCNCPoint1[11365] = {X 202.7154, Y 21.7361, Z -1.3333, A 0.000, B 0.000, C 0.000 }
gfCNCPoint1[11366] = {X 202.6050, Y 23.4182, Z -1.3333, A 0.000, B 0.000, C 0.000 }
gfCNCPoint1[11367] = {X 202.3029, Y 25.0766, Z -1.3333, A 0.000, B 0.000, C 0.000 }
gfCNCPoint1[11368] = {X 201.8255, Y 26.6078, Z -1.3333, A 0.000, B 0.000, C 0.000 }
gfCNCPoint1[11369] = {X 201.1373, Y 28.0566, Z -1.3333, A 0.000, B 0.000, C 0.000 }
gfCNCPoint1[11370] = {X 200.2522, Y 29.3941, Z -1.3333, A 0.000, B 0.000, C 0.000 }
gfCNCPoint1[11371] = {X 199.1876, Y 30.5938, Z -1.3333, A 0.000, B 0.000, C 0.000 }
gfCNCPoint1[11372] = {X 197.9648, Y 31.6317, Z -1.3333, A 0.000, B 0.000, C 0.000 }
gfCNCPoint1[11373] = {X 198.7269, Y 31.8155, Z -1.3333, A 0.000, B 0.000, C 0.000 }
gfCNCPoint1[11374] = {X 199.4385, Y 32.1444, Z -1.3333, A 0.000, B 0.000, C 0.000 }
gfCNCPoint1[11375] = {X 200.0723, Y 32.6058, Z -1.3333, A 0.000, B 0.000, C 0.000 }
gfCNCPoint1[11376] = {X 200.6039, Y 33.1820, Z -1.3333, A 0.000, B 0.000, C 0.000 }
gfCNCPoint1[11377] = {X 201.0129, Y 33.8507, Z -1.3333, A 0.000, B 0.000, C 0.000 }
gfCNCPoint1[11378] = {X 204.0341, Y 40.0925, Z -1.3333, A 0.000, B 0.000, C 0.000 }
gfCNCPoint1[11379] = {X 204.3309, Y 40.9342, Z -1.3333, A 0.000, B 0.000, C 0.000 }
gfCNCPoint1[11380] = {X 204.4337, Y 41.8209, Z -1.3333, A 0.000, B 0.000, C 0.000 }
gfCNCPoint1[11381] = {X 204.3373, Y 42.7082, Z -1.3333, A 0.000, B 0.000, C 0.000 }
gfCNCPoint1[11382] = {X 204.0465, Y 43.5521, Z -1.3333, A 0.000, B 0.000, C 0.000 }
gfCNCPoint1[11383] = {X 203.5758, Y 44.3105, Z -1.3333, A 0.000, B 0.000, C 0.000 }
gfCNCPoint1[11384] = {X 202.9487, Y 44.9456, Z -1.3333, A 0.000, B 0.000, C 0.000 }
gfCNCPoint1[11385] = {X 202.4125, Y 45.3791, Z -1.3333, A 0.000, B 0.000, C 0.000 }
gfCNCPoint1[11386] = {X 201.7354, Y 45.8207, Z -1.3333, A 0.000, B 0.000, C 0.000 }
gfCNCPoint1[11387] = {X 200.9837, Y 46.1178, Z -1.3333, A 0.000, B 0.000, C 0.000 }
gfCNCPoint1[11388] = {X 200.1876, Y 46.2583, Z -1.3333, A 0.000, B 0.000, C 0.000 }
gfCNCPoint1[11389] = {X 199.3795, Y 46.2366, Z -1.3333, A 0.000, B 0.000, C 0.000 }
gfCNCPoint1[11390] = {X 198.5922, Y 46.0536, Z -1.3333, A 0.000, B 0.000, C 0.000 }
gfCNCPoint1[11391] = {X 196.9033, Y 46.9629, Z -1.3333, A 0.000, B 0.000, C 0.000 }
gfCNCPoint1[11392] = {X 195.1556, Y 47.7531, Z -1.3333, A 0.000, B 0.000, C 0.000 }
gfCNCPoint1[11393] = {X 193.3575, Y 48.4206, Z -1.3333, A 0.000, B 0.000, C 0.000 }
gfCNCPoint1[11394] = {X 192.7968, Y 48.6154, Z -1.3333, A 0.000, B 0.000, C 0.000 }
gfCNCPoint1[11395] = {X 190.6042, Y 49.1997, Z -1.3333, A 0.000, B 0.000, C 0.000 }
gfCNCPoint1[11396] = {X 188.3638, Y 49.5606, Z -1.3333, A 0.000, B 0.000, C 0.000 }
gfCNCPoint1[11397] = {X 186.0986, Y 49.6943, Z -1.3333, A 0.000, B 0.000, C 0.000 }
gfCNCPoint1[11398] = {X 183.8314, Y 49.5995, Z -1.3333, A 0.000, B 0.000, C 0.000 }
gfCNCPoint1[11399] = {X 181.5852, Y 49.2772, Z -1.3333, A 0.000, B 0.000, C 0.000 }
gfCNCPoint1[11400] = {X 179.7338, Y 48.8145, Z -1.3333, A 0.000, B 0.000, C 0.000 }
gfCNCPoint1[11401] = {X 177.9472, Y 48.1438, Z -1.3333, A 0.000, B 0.000, C 0.000 }
gfCNCPoint1[11402] = {X 176.2487, Y 47.2738, Z -1.3333, A 0.000, B 0.000, C 0.000 }
gfCNCPoint1[11403] = {X 174.6604, Y 46.2159, Z -1.3333, A 0.000, B 0.000, C 0.000 }
gfCNCPoint1[11404] = {X 173.4569, Y 45.2001, Z -1.3333, A 0.000, B 0.000, C 0.000 }
gfCNCPoint1[11405] = {X 172.3860, Y 44.0454, Z -1.3333, A 0.000, B 0.000, C 0.000 }
gfCNCPoint1[11406] = {X 171.4636, Y 42.7689, Z -1.3333, A 0.000, B 0.000, C 0.000 }
gfCNCPoint1[11407] = {X 170.7035, Y 41.3896, Z -1.3333, A 0.000, B 0.000, C 0.000 }
gfCNCPoint1[11408] = {X 170.1169, Y 39.9280, Z -1.3333, A 0.000, B 0.000, C 0.000 }
gfCNCPoint1[11409] = {X 169.7126, Y 38.4059, Z -1.3333, A 0.000, B 0.000, C 0.000 }
gfCNCPoint1[11410] = {X 169.4966, Y 36.8460, Z -1.3333, A 0.000, B 0.000, C 0.000 }
gfCNCPoint1[11411] = {X 169.4135, Y 35.0509, Z -1.3333, A 0.000, B 0.000, C 0.000 }
gfCNCPoint1[11412] = {X 169.5560, Y 33.2595, Z -1.3333, A 0.000, B 0.000, C 0.000 }
gfCNCPoint1[11413] = {X 169.9219, Y 31.5001, Z -1.3333, A 0.000, B 0.000, C 0.000 }
gfCNCPoint1[11414] = {X 170.5055, Y 29.8005, Z -1.3333, A 0.000, B 0.000, C 0.000 }
gfCNCPoint1[11415] = {X 171.2086, Y 28.3902, Z -1.3333, A 0.000, B 0.000, C 0.000 }
gfCNCPoint1[11416] = {X 172.1140, Y 27.1004, Z -1.3333, A 0.000, B 0.000, C 0.000 }
gfCNCPoint1[11417] = {X 173.2015, Y 25.9600, Z -1.3333, A 0.000, B 0.000, C 0.000 }
gfCNCPoint1[11418] = {X 174.4467, Y 24.9943, Z -1.3333, A 0.000, B 0.000, C 0.000 }
gfCNCPoint1[11419] = {X 175.8220, Y 24.2249, Z -1.3333, A 0.000, B 0.000, C 0.000 }
gfCNCPoint1[11420] = {X 175.0309, Y 24.0141, Z -1.3333, A 0.000, B 0.000, C 0.000 }
gfCNCPoint1[11421] = {X 174.2992, Y 23.6465, Z -1.3333, A 0.000, B 0.000, C 0.000 }
gfCNCPoint1[11422] = {X 173.6578, Y 23.1377, Z -1.3333, A 0.000, B 0.000, C 0.000 }
gfCNCPoint1[11423] = {X 173.1333, Y 22.5089, Z -1.3333, A 0.000, B 0.000, C 0.000 }
gfCNCPoint1[11424] = {X 172.7479, Y 21.7866, Z -1.3333, A 0.000, B 0.000, C 0.000 }
gfCNCPoint1[11425] = {X 171.4542, Y 18.6179, Z -1.3333, A 0.000, B 0.000, C 0.000 }
gfCNCPoint1[11426] = {X 167.6769, Y 20.1601, Z -1.3333, A 0.000, B 0.000, C 0.000 }
gfCNCPoint1[11427] = {X 167.6769, Y 20.1601, Z 1.6667, A 0.000, B 0.000, C 0.000 }
gfCNCPoint1[11428] = {X 167.6769, Y 20.1601, Z 11.0000, A 0.000, B 0.000, C 0.000 }
gfCNCPoint1[11429] = {X 210.1662, Y 28.5743, Z 11.0000, A 0.000, B 0.000, C 0.000 }
gfCNCPoint1[11430] = {X 210.1662, Y 28.5743, Z 1.6667, A 0.000, B 0.000, C 0.000 }
gfCNCPoint1[11431] = {X 210.1662, Y 28.5743, Z -1.3333, A 0.000, B 0.000, C 0.000 }
gfCNCPoint1[11432] = {X 214.2462, Y 28.5743, Z -1.3333, A 0.000, B 0.000, C 0.000 }
gfCNCPoint1[11433] = {X 214.2462, Y 17.4624, Z -1.3333, A 0.000, B 0.000, C 0.000 }
gfCNCPoint1[11434] = {X 214.2409, Y 16.7694, Z -1.3333, A 0.000, B 0.000, C 0.000 }
gfCNCPoint1[11435] = {X 214.2436, Y 16.2733, Z -1.3333, A 0.000, B 0.000, C 0.000 }
gfCNCPoint1[11436] = {X 213.6053, Y 15.6021, Z -1.3333, A 0.000, B 0.000, C 0.000 }
gfCNCPoint1[11437] = {X 213.1248, Y 14.8103, Z -1.3333, A 0.000, B 0.000, C 0.000 }
gfCNCPoint1[11438] = {X 212.8242, Y 13.9342, Z -1.3333, A 0.000, B 0.000, C 0.000 }
gfCNCPoint1[11439] = {X 212.7172, Y 13.0141, Z -1.3333, A 0.000, B 0.000, C 0.000 }
gfCNCPoint1[11440] = {X 212.7170, Y 12.1868, Z -1.3333, A 0.000, B 0.000, C 0.000 }
gfCNCPoint1[11441] = {X 212.8253, Y 11.2255, Z -1.3333, A 0.000, B 0.000, C 0.000 }
gfCNCPoint1[11442] = {X 213.1448, Y 10.3124, Z -1.3333, A 0.000, B 0.000, C 0.000 }
gfCNCPoint1[11443] = {X 213.6595, Y 9.4933, Z -1.3333, A 0.000, B 0.000, C 0.000 }
gfCNCPoint1[11444] = {X 214.3435, Y 8.8093, Z -1.3333, A 0.000, B 0.000, C 0.000 }
gfCNCPoint1[11445] = {X 215.1626, Y 8.2946, Z -1.3333, A 0.000, B 0.000, C 0.000 }
gfCNCPoint1[11446] = {X 216.0757, Y 7.9751, Z -1.3333, A 0.000, B 0.000, C 0.000 }
gfCNCPoint1[11447] = {X 217.0370, Y 7.8668, Z -1.3333, A 0.000, B 0.000, C 0.000 }
gfCNCPoint1[11448] = {X 223.4805, Y 7.8668, Z -1.3333, A 0.000, B 0.000, C 0.000 }
gfCNCPoint1[11449] = {X 224.4418, Y 7.9751, Z -1.3333, A 0.000, B 0.000, C 0.000 }
gfCNCPoint1[11450] = {X 225.3549, Y 8.2946, Z -1.3333, A 0.000, B 0.000, C 0.000 }
gfCNCPoint1[11451] = {X 226.1740, Y 8.8093, Z -1.3333, A 0.000, B 0.000, C 0.000 }
gfCNCPoint1[11452] = {X 226.8580, Y 9.4933, Z -1.3333, A 0.000, B 0.000, C 0.000 }
gfCNCPoint1[11453] = {X 227.3727, Y 10.3124, Z -1.3333, A 0.000, B 0.000, C 0.000 }
gfCNCPoint1[11454] = {X 227.6922, Y 11.2255, Z -1.3333, A 0.000, B 0.000, C 0.000 }
gfCNCPoint1[11455] = {X 227.8005, Y 12.1868, Z -1.3333, A 0.000, B 0.000, C 0.000 }
gfCNCPoint1[11456] = {X 227.8005, Y 12.9781, Z -1.3333, A 0.000, B 0.000, C 0.000 }
gfCNCPoint1[11457] = {X 227.6991, Y 13.9084, Z -1.3333, A 0.000, B 0.000, C 0.000 }
gfCNCPoint1[11458] = {X 227.3998, Y 14.7951, Z -1.3333, A 0.000, B 0.000, C 0.000 }
gfCNCPoint1[11459] = {X 226.9165, Y 15.5964, Z -1.3333, A 0.000, B 0.000, C 0.000 }
gfCNCPoint1[11460] = {X 226.2720, Y 16.2749, Z -1.3333, A 0.000, B 0.000, C 0.000 }
gfCNCPoint1[11461] = {X 226.2729, Y 40.9153, Z -1.3333, A 0.000, B 0.000, C 0.000 }
gfCNCPoint1[11462] = {X 226.9106, Y 41.5853, Z -1.3333, A 0.000, B 0.000, C 0.000 }
gfCNCPoint1[11463] = {X 227.3910, Y 42.3757, Z -1.3333, A 0.000, B 0.000, C 0.000 }
gfCNCPoint1[11464] = {X 227.6922, Y 43.2502, Z -1.3333, A 0.000, B 0.000, C 0.000 }
gfCNCPoint1[11465] = {X 227.8003, Y 44.1689, Z -1.3333, A 0.000, B 0.000, C 0.000 }
gfCNCPoint1[11466] = {X 227.8005, Y 45.0000, Z -1.3333, A 0.000, B 0.000, C 0.000 }
gfCNCPoint1[11467] = {X 227.6922, Y 45.9613, Z -1.3333, A 0.000, B 0.000, C 0.000 }
gfCNCPoint1[11468] = {X 227.3727, Y 46.8744, Z -1.3333, A 0.000, B 0.000, C 0.000 }
gfCNCPoint1[11469] = {X 226.8580, Y 47.6935, Z -1.3333, A 0.000, B 0.000, C 0.000 }
gfCNCPoint1[11470] = {X 226.1740, Y 48.3775, Z -1.3333, A 0.000, B 0.000, C 0.000 }
gfCNCPoint1[11471] = {X 225.3549, Y 48.8922, Z -1.3333, A 0.000, B 0.000, C 0.000 }
gfCNCPoint1[11472] = {X 224.4418, Y 49.2117, Z -1.3333, A 0.000, B 0.000, C 0.000 }
gfCNCPoint1[11473] = {X 223.4805, Y 49.3200, Z -1.3333, A 0.000, B 0.000, C 0.000 }
gfCNCPoint1[11474] = {X 217.0370, Y 49.3200, Z -1.3333, A 0.000, B 0.000, C 0.000 }
gfCNCPoint1[11475] = {X 216.0805, Y 49.2128, Z -1.3333, A 0.000, B 0.000, C 0.000 }
gfCNCPoint1[11476] = {X 215.1715, Y 48.8964, Z -1.3333, A 0.000, B 0.000, C 0.000 }
gfCNCPoint1[11477] = {X 214.3551, Y 48.3867, Z -1.3333, A 0.000, B 0.000, C 0.000 }
gfCNCPoint1[11478] = {X 213.6718, Y 47.7088, Z -1.3333, A 0.000, B 0.000, C 0.000 }
gfCNCPoint1[11479] = {X 213.1556, Y 46.8965, Z -1.3333, A 0.000, B 0.000, C 0.000 }
gfCNCPoint1[11480] = {X 212.8320, Y 45.9901, Z -1.3333, A 0.000, B 0.000, C 0.000 }
gfCNCPoint1[11481] = {X 212.7172, Y 45.0345, Z -1.3333, A 0.000, B 0.000, C 0.000 }
gfCNCPoint1[11482] = {X 212.7170, Y 44.2008, Z -1.3333, A 0.000, B 0.000, C 0.000 }
gfCNCPoint1[11483] = {X 212.7890, Y 43.4209, Z -1.3333, A 0.000, B 0.000, C 0.000 }
gfCNCPoint1[11484] = {X 213.0026, Y 42.6674, Z -1.3333, A 0.000, B 0.000, C 0.000 }
gfCNCPoint1[11485] = {X 213.3504, Y 41.9658, Z -1.3333, A 0.000, B 0.000, C 0.000 }
gfCNCPoint1[11486] = {X 213.8209, Y 41.3396, Z -1.3333, A 0.000, B 0.000, C 0.000 }
gfCNCPoint1[11487] = {X 214.2418, Y 40.8754, Z -1.3333, A 0.000, B 0.000, C 0.000 }
gfCNCPoint1[11488] = {X 214.2462, Y 40.3062, Z -1.3333, A 0.000, B 0.000, C 0.000 }
gfCNCPoint1[11489] = {X 214.2462, Y 28.5743, Z -1.3333, A 0.000, B 0.000, C 0.000 }
gfCNCPoint1[11490] = {X 210.2462, Y 28.5743, Z -1.3333, A 0.000, B 0.000, C 0.000 }
gfCNCPoint1[11491] = {X 214.3262, Y 28.5743, Z -1.3333, A 0.000, B 0.000, C 0.000 }
gfCNCPoint1[11492] = {X 214.3262, Y 17.4621, Z -1.3333, A 0.000, B 0.000, C 0.000 }
gfCNCPoint1[11493] = {X 214.3209, Y 16.7693, Z -1.3333, A 0.000, B 0.000, C 0.000 }
gfCNCPoint1[11494] = {X 214.3238, Y 16.2362, Z -1.3333, A 0.000, B 0.000, C 0.000 }
gfCNCPoint1[11495] = {X 213.6859, Y 15.5756, Z -1.3333, A 0.000, B 0.000, C 0.000 }
gfCNCPoint1[11496] = {X 213.2052, Y 14.7931, Z -1.3333, A 0.000, B 0.000, C 0.000 }
gfCNCPoint1[11497] = {X 212.9042, Y 13.9255, Z -1.3333, A 0.000, B 0.000, C 0.000 }
gfCNCPoint1[11498] = {X 212.7972, Y 13.0135, Z -1.3333, A 0.000, B 0.000, C 0.000 }
gfCNCPoint1[11499] = {X 212.7970, Y 12.1868, Z -1.3333, A 0.000, B 0.000, C 0.000 }
gfCNCPoint1[11500] = {X 212.9033, Y 11.2433, Z -1.3333, A 0.000, B 0.000, C 0.000 }
gfCNCPoint1[11501] = {X 213.2169, Y 10.3472, Z -1.3333, A 0.000, B 0.000, C 0.000 }
gfCNCPoint1[11502] = {X 213.7220, Y 9.5432, Z -1.3333, A 0.000, B 0.000, C 0.000 }
gfCNCPoint1[11503] = {X 214.3934, Y 8.8719, Z -1.3333, A 0.000, B 0.000, C 0.000 }
gfCNCPoint1[11504] = {X 215.1973, Y 8.3667, Z -1.3333, A 0.000, B 0.000, C 0.000 }
gfCNCPoint1[11505] = {X 216.0935, Y 8.0531, Z -1.3333, A 0.000, B 0.000, C 0.000 }
gfCNCPoint1[11506] = {X 217.0370, Y 7.9468, Z -1.3333, A 0.000, B 0.000, C 0.000 }
gfCNCPoint1[11507] = {X 223.4805, Y 7.9468, Z -1.3333, A 0.000, B 0.000, C 0.000 }
gfCNCPoint1[11508] = {X 224.4240, Y 8.0531, Z -1.3333, A 0.000, B 0.000, C 0.000 }
gfCNCPoint1[11509] = {X 225.3201, Y 8.3667, Z -1.3333, A 0.000, B 0.000, C 0.000 }
gfCNCPoint1[11510] = {X 226.1241, Y 8.8718, Z -1.3333, A 0.000, B 0.000, C 0.000 }
gfCNCPoint1[11511] = {X 226.7954, Y 9.5432, Z -1.3333, A 0.000, B 0.000, C 0.000 }
gfCNCPoint1[11512] = {X 227.3006, Y 10.3471, Z -1.3333, A 0.000, B 0.000, C 0.000 }
gfCNCPoint1[11513] = {X 227.6142, Y 11.2433, Z -1.3333, A 0.000, B 0.000, C 0.000 }
gfCNCPoint1[11514] = {X 227.7205, Y 12.1868, Z -1.3333, A 0.000, B 0.000, C 0.000 }
gfCNCPoint1[11515] = {X 227.7205, Y 12.9781, Z -1.3333, A 0.000, B 0.000, C 0.000 }
gfCNCPoint1[11516] = {X 227.6190, Y 13.9002, Z -1.3333, A 0.000, B 0.000, C 0.000 }
gfCNCPoint1[11517] = {X 227.3194, Y 14.7781, Z -1.3333, A 0.000, B 0.000, C 0.000 }
gfCNCPoint1[11518] = {X 226.8360, Y 15.5699, Z -1.3333, A 0.000, B 0.000, C 0.000 }
gfCNCPoint1[11519] = {X 226.1920, Y 16.2376, Z -1.3333, A 0.000, B 0.000, C 0.000 }
gfCNCPoint1[11520] = {X 226.1929, Y 40.9526, Z -1.3333, A 0.000, B 0.000, C 0.000 }
gfCNCPoint1[11521] = {X 226.8302, Y 41.6120, Z -1.3333, A 0.000, B 0.000, C 0.000 }
gfCNCPoint1[11522] = {X 227.3107, Y 42.3930, Z -1.3333, A 0.000, B 0.000, C 0.000 }
gfCNCPoint1[11523] = {X 227.6122, Y 43.2590, Z -1.3333, A 0.000, B 0.000, C 0.000 }
gfCNCPoint1[11524] = {X 227.7203, Y 44.1697, Z -1.3333, A 0.000, B 0.000, C 0.000 }
gfCNCPoint1[11525] = {X 227.7205, Y 45.0000, Z -1.3333, A 0.000, B 0.000, C 0.000 }
gfCNCPoint1[11526] = {X 227.6142, Y 45.9435, Z -1.3333, A 0.000, B 0.000, C 0.000 }
gfCNCPoint1[11527] = {X 227.3006, Y 46.8397, Z -1.3333, A 0.000, B 0.000, C 0.000 }
gfCNCPoint1[11528] = {X 226.7954, Y 47.6436, Z -1.3333, A 0.000, B 0.000, C 0.000 }
gfCNCPoint1[11529] = {X 226.1241, Y 48.3150, Z -1.3333, A 0.000, B 0.000, C 0.000 }
gfCNCPoint1[11530] = {X 225.3201, Y 48.8201, Z -1.3333, A 0.000, B 0.000, C 0.000 }
gfCNCPoint1[11531] = {X 224.4240, Y 49.1337, Z -1.3333, A 0.000, B 0.000, C 0.000 }
gfCNCPoint1[11532] = {X 223.4805, Y 49.2400, Z -1.3333, A 0.000, B 0.000, C 0.000 }
gfCNCPoint1[11533] = {X 217.0370, Y 49.2400, Z -1.3333, A 0.000, B 0.000, C 0.000 }
gfCNCPoint1[11534] = {X 216.0982, Y 49.1348, Z -1.3333, A 0.000, B 0.000, C 0.000 }
gfCNCPoint1[11535] = {X 215.2061, Y 48.8243, Z -1.3333, A 0.000, B 0.000, C 0.000 }
gfCNCPoint1[11536] = {X 214.4048, Y 48.3240, Z -1.3333, A 0.000, B 0.000, C 0.000 }
gfCNCPoint1[11537] = {X 213.7341, Y 47.6587, Z -1.3333, A 0.000, B 0.000, C 0.000 }
gfCNCPoint1[11538] = {X 213.2275, Y 46.8614, Z -1.3333, A 0.000, B 0.000, C 0.000 }
gfCNCPoint1[11539] = {X 212.9099, Y 45.9717, Z -1.3333, A 0.000, B 0.000, C 0.000 }
gfCNCPoint1[11540] = {X 212.7972, Y 45.0338, Z -1.3333, A 0.000, B 0.000, C 0.000 }
gfCNCPoint1[11541] = {X 212.7970, Y 44.2008, Z -1.3333, A 0.000, B 0.000, C 0.000 }
gfCNCPoint1[11542] = {X 212.8677, Y 43.4356, Z -1.3333, A 0.000, B 0.000, C 0.000 }
gfCNCPoint1[11543] = {X 213.0772, Y 42.6962, Z -1.3333, A 0.000, B 0.000, C 0.000 }
gfCNCPoint1[11544] = {X 213.4185, Y 42.0077, Z -1.3333, A 0.000, B 0.000, C 0.000 }
gfCNCPoint1[11545] = {X 213.8802, Y 41.3934, Z -1.3333, A 0.000, B 0.000, C 0.000 }
gfCNCPoint1[11546] = {X 214.3216, Y 40.9065, Z -1.3333, A 0.000, B 0.000, C 0.000 }
gfCNCPoint1[11547] = {X 214.3262, Y 40.3065, Z -1.3333, A 0.000, B 0.000, C 0.000 }
gfCNCPoint1[11548] = {X 214.3262, Y 28.5743, Z -1.3333, A 0.000, B 0.000, C 0.000 }
gfCNCPoint1[11549] = {X 210.3262, Y 28.5743, Z -1.3333, A 0.000, B 0.000, C 0.000 }
gfCNCPoint1[11550] = {X 214.4062, Y 28.5743, Z -1.3333, A 0.000, B 0.000, C 0.000 }
gfCNCPoint1[11551] = {X 214.4062, Y 17.4617, Z -1.3333, A 0.000, B 0.000, C 0.000 }
gfCNCPoint1[11552] = {X 214.4009, Y 16.7692, Z -1.3333, A 0.000, B 0.000, C 0.000 }
gfCNCPoint1[11553] = {X 214.4040, Y 16.1987, Z -1.3333, A 0.000, B 0.000, C 0.000 }
gfCNCPoint1[11554] = {X 213.7665, Y 15.5488, Z -1.3333, A 0.000, B 0.000, C 0.000 }
gfCNCPoint1[11555] = {X 213.2856, Y 14.7759, Z -1.3333, A 0.000, B 0.000, C 0.000 }
gfCNCPoint1[11556] = {X 212.9843, Y 13.9168, Z -1.3333, A 0.000, B 0.000, C 0.000 }
gfCNCPoint1[11557] = {X 212.8772, Y 13.0128, Z -1.3333, A 0.000, B 0.000, C 0.000 }
gfCNCPoint1[11558] = {X 212.8770, Y 12.1868, Z -1.3333, A 0.000, B 0.000, C 0.000 }
gfCNCPoint1[11559] = {X 212.9813, Y 11.2611, Z -1.3333, A 0.000, B 0.000, C 0.000 }
gfCNCPoint1[11560] = {X 213.2890, Y 10.3819, Z -1.3333, A 0.000, B 0.000, C 0.000 }
gfCNCPoint1[11561] = {X 213.7846, Y 9.5931, Z -1.3333, A 0.000, B 0.000, C 0.000 }
gfCNCPoint1[11562] = {X 214.4433, Y 8.9344, Z -1.3333, A 0.000, B 0.000, C 0.000 }
gfCNCPoint1[11563] = {X 215.2321, Y 8.4388, Z -1.3333, A 0.000, B 0.000, C 0.000 }
gfCNCPoint1[11564] = {X 216.1113, Y 8.1311, Z -1.3333, A 0.000, B 0.000, C 0.000 }
gfCNCPoint1[11565] = {X 217.0370, Y 8.0268, Z -1.3333, A 0.000, B 0.000, C 0.000 }
gfCNCPoint1[11566] = {X 223.4805, Y 8.0268, Z -1.3333, A 0.000, B 0.000, C 0.000 }
gfCNCPoint1[11567] = {X 224.4062, Y 8.1311, Z -1.3333, A 0.000, B 0.000, C 0.000 }
gfCNCPoint1[11568] = {X 225.2854, Y 8.4388, Z -1.3333, A 0.000, B 0.000, C 0.000 }
gfCNCPoint1[11569] = {X 226.0742, Y 8.9344, Z -1.3333, A 0.000, B 0.000, C 0.000 }
gfCNCPoint1[11570] = {X 226.7329, Y 9.5931, Z -1.3333, A 0.000, B 0.000, C 0.000 }
gfCNCPoint1[11571] = {X 227.2285, Y 10.3819, Z -1.3333, A 0.000, B 0.000, C 0.000 }
gfCNCPoint1[11572] = {X 227.5362, Y 11.2611, Z -1.3333, A 0.000, B 0.000, C 0.000 }
gfCNCPoint1[11573] = {X 227.6405, Y 12.1868, Z -1.3333, A 0.000, B 0.000, C 0.000 }
gfCNCPoint1[11574] = {X 227.6405, Y 12.9781, Z -1.3333, A 0.000, B 0.000, C 0.000 }
gfCNCPoint1[11575] = {X 227.5389, Y 13.8919, Z -1.3333, A 0.000, B 0.000, C 0.000 }
gfCNCPoint1[11576] = {X 227.2390, Y 14.7611, Z -1.3333, A 0.000, B 0.000, C 0.000 }
gfCNCPoint1[11577] = {X 226.7555, Y 15.5431, Z -1.3333, A 0.000, B 0.000, C 0.000 }
gfCNCPoint1[11578] = {X 226.1120, Y 16.1999, Z -1.3333, A 0.000, B 0.000, C 0.000 }
gfCNCPoint1[11579] = {X 226.1129, Y 40.9903, Z -1.3333, A 0.000, B 0.000, C 0.000 }
gfCNCPoint1[11580] = {X 226.7497, Y 41.6390, Z -1.3333, A 0.000, B 0.000, C 0.000 }
gfCNCPoint1[11581] = {X 227.2304, Y 42.4104, Z -1.3333, A 0.000, B 0.000, C 0.000 }
gfCNCPoint1[11582] = {X 227.5321, Y 43.2679, Z -1.3333, A 0.000, B 0.000, C 0.000 }
gfCNCPoint1[11583] = {X 227.6403, Y 44.1704, Z -1.3333, A 0.000, B 0.000, C 0.000 }
gfCNCPoint1[11584] = {X 227.6405, Y 45.0000, Z -1.3333, A 0.000, B 0.000, C 0.000 }
gfCNCPoint1[11585] = {X 227.5362, Y 45.9257, Z -1.3333, A 0.000, B 0.000, C 0.000 }
gfCNCPoint1[11586] = {X 227.2285, Y 46.8050, Z -1.3333, A 0.000, B 0.000, C 0.000 }
gfCNCPoint1[11587] = {X 226.7329, Y 47.5937, Z -1.3333, A 0.000, B 0.000, C 0.000 }
gfCNCPoint1[11588] = {X 226.0742, Y 48.2524, Z -1.3333, A 0.000, B 0.000, C 0.000 }
gfCNCPoint1[11589] = {X 225.2854, Y 48.7480, Z -1.3333, A 0.000, B 0.000, C 0.000 }
gfCNCPoint1[11590] = {X 224.4062, Y 49.0557, Z -1.3333, A 0.000, B 0.000, C 0.000 }
gfCNCPoint1[11591] = {X 223.4805, Y 49.1600, Z -1.3333, A 0.000, B 0.000, C 0.000 }
gfCNCPoint1[11592] = {X 217.0370, Y 49.1600, Z -1.3333, A 0.000, B 0.000, C 0.000 }
gfCNCPoint1[11593] = {X 216.1160, Y 49.0568, Z -1.3333, A 0.000, B 0.000, C 0.000 }
gfCNCPoint1[11594] = {X 215.2406, Y 48.7521, Z -1.3333, A 0.000, B 0.000, C 0.000 }
gfCNCPoint1[11595] = {X 214.4544, Y 48.2613, Z -1.3333, A 0.000, B 0.000, C 0.000 }
gfCNCPoint1[11596] = {X 213.7965, Y 47.6085, Z -1.3333, A 0.000, B 0.000, C 0.000 }
gfCNCPoint1[11597] = {X 213.2993, Y 46.8263, Z -1.3333, A 0.000, B 0.000, C 0.000 }
gfCNCPoint1[11598] = {X 212.9877, Y 45.9534, Z -1.3333, A 0.000, B 0.000, C 0.000 }
gfCNCPoint1[11599] = {X 212.8771, Y 45.0332, Z -1.3333, A 0.000, B 0.000, C 0.000 }
gfCNCPoint1[11600] = {X 212.8770, Y 44.2008, Z -1.3333, A 0.000, B 0.000, C 0.000 }
gfCNCPoint1[11601] = {X 212.9463, Y 43.4502, Z -1.3333, A 0.000, B 0.000, C 0.000 }
gfCNCPoint1[11602] = {X 213.1518, Y 42.7250, Z -1.3333, A 0.000, B 0.000, C 0.000 }
gfCNCPoint1[11603] = {X 213.4867, Y 42.0497, Z -1.3333, A 0.000, B 0.000, C 0.000 }
gfCNCPoint1[11604] = {X 213.9394, Y 41.4471, Z -1.3333, A 0.000, B 0.000, C 0.000 }
gfCNCPoint1[11605] = {X 214.4013, Y 40.9376, Z -1.3333, A 0.000, B 0.000, C 0.000 }
gfCNCPoint1[11606] = {X 214.4062, Y 40.3069, Z -1.3333, A 0.000, B 0.000, C 0.000 }
gfCNCPoint1[11607] = {X 214.4062, Y 28.5743, Z -1.3333, A 0.000, B 0.000, C 0.000 }
gfCNCPoint1[11608] = {X 210.4062, Y 28.5743, Z -1.3333, A 0.000, B 0.000, C 0.000 }
gfCNCPoint1[11609] = {X 214.4862, Y 28.5743, Z -1.3333, A 0.000, B 0.000, C 0.000 }
gfCNCPoint1[11610] = {X 214.4862, Y 17.4614, Z -1.3333, A 0.000, B 0.000, C 0.000 }
gfCNCPoint1[11611] = {X 214.4809, Y 16.7691, Z -1.3333, A 0.000, B 0.000, C 0.000 }
gfCNCPoint1[11612] = {X 214.4842, Y 16.1607, Z -1.3333, A 0.000, B 0.000, C 0.000 }
gfCNCPoint1[11613] = {X 214.4264, Y 16.1135, Z -1.3333, A 0.000, B 0.000, C 0.000 }
gfCNCPoint1[11614] = {X 214.3695, Y 16.0652, Z -1.3333, A 0.000, B 0.000, C 0.000 }
gfCNCPoint1[11615] = {X 213.7785, Y 15.4333, Z -1.3333, A 0.000, B 0.000, C 0.000 }
gfCNCPoint1[11616] = {X 213.3340, Y 14.6910, Z -1.3333, A 0.000, B 0.000, C 0.000 }
gfCNCPoint1[11617] = {X 213.0561, Y 13.8717, Z -1.3333, A 0.000, B 0.000, C 0.000 }
gfCNCPoint1[11618] = {X 212.9572, Y 13.0121, Z -1.3333, A 0.000, B 0.000, C 0.000 }
gfCNCPoint1[11619] = {X 212.9570, Y 12.1868, Z -1.3333, A 0.000, B 0.000, C 0.000 }
gfCNCPoint1[11620] = {X 213.0593, Y 11.2789, Z -1.3333, A 0.000, B 0.000, C 0.000 }
gfCNCPoint1[11621] = {X 213.3611, Y 10.4166, Z -1.3333, A 0.000, B 0.000, C 0.000 }
gfCNCPoint1[11622] = {X 213.8471, Y 9.6430, Z -1.3333, A 0.000, B 0.000, C 0.000 }
gfCNCPoint1[11623] = {X 214.4932, Y 8.9969, Z -1.3333, A 0.000, B 0.000, C 0.000 }
gfCNCPoint1[11624] = {X 215.2668, Y 8.5109, Z -1.3333, A 0.000, B 0.000, C 0.000 }
gfCNCPoint1[11625] = {X 216.1291, Y 8.2091, Z -1.3333, A 0.000, B 0.000, C 0.000 }
gfCNCPoint1[11626] = {X 217.0370, Y 8.1068, Z -1.3333, A 0.000, B 0.000, C 0.000 }
gfCNCPoint1[11627] = {X 223.4805, Y 8.1068, Z -1.3333, A 0.000, B 0.000, C 0.000 }
gfCNCPoint1[11628] = {X 224.3884, Y 8.2091, Z -1.3333, A 0.000, B 0.000, C 0.000 }
gfCNCPoint1[11629] = {X 225.2507, Y 8.5109, Z -1.3333, A 0.000, B 0.000, C 0.000 }
gfCNCPoint1[11630] = {X 226.0243, Y 8.9969, Z -1.3333, A 0.000, B 0.000, C 0.000 }
gfCNCPoint1[11631] = {X 226.6704, Y 9.6430, Z -1.3333, A 0.000, B 0.000, C 0.000 }
gfCNCPoint1[11632] = {X 227.1564, Y 10.4166, Z -1.3333, A 0.000, B 0.000, C 0.000 }
gfCNCPoint1[11633] = {X 227.4582, Y 11.2789, Z -1.3333, A 0.000, B 0.000, C 0.000 }
gfCNCPoint1[11634] = {X 227.5605, Y 12.1868, Z -1.3333, A 0.000, B 0.000, C 0.000 }
gfCNCPoint1[11635] = {X 227.5605, Y 12.9781, Z -1.3333, A 0.000, B 0.000, C 0.000 }
gfCNCPoint1[11636] = {X 227.4587, Y 13.8836, Z -1.3333, A 0.000, B 0.000, C 0.000 }
gfCNCPoint1[11637] = {X 227.1586, Y 14.7439, Z -1.3333, A 0.000, B 0.000, C 0.000 }
gfCNCPoint1[11638] = {X 226.6750, Y 15.5161, Z -1.3333, A 0.000, B 0.000, C 0.000 }
gfCNCPoint1[11639] = {X 226.0320, Y 16.1617, Z -1.3333, A 0.000, B 0.000, C 0.000 }
gfCNCPoint1[11640] = {X 226.0329, Y 41.0286, Z -1.3333, A 0.000, B 0.000, C 0.000 }
gfCNCPoint1[11641] = {X 226.1408, Y 41.1154, Z -1.3333, A 0.000, B 0.000, C 0.000 }
gfCNCPoint1[11642] = {X 226.7342, Y 41.7471, Z -1.3333, A 0.000, B 0.000, C 0.000 }
gfCNCPoint1[11643] = {X 227.1807, Y 42.4899, Z -1.3333, A 0.000, B 0.000, C 0.000 }
gfCNCPoint1[11644] = {X 227.4603, Y 43.3103, Z -1.3333, A 0.000, B 0.000, C 0.000 }
gfCNCPoint1[11645] = {X 227.5603, Y 44.1712, Z -1.3333, A 0.000, B 0.000, C 0.000 }
gfCNCPoint1[11646] = {X 227.5605, Y 45.0000, Z -1.3333, A 0.000, B 0.000, C 0.000 }
gfCNCPoint1[11647] = {X 227.4582, Y 45.9079, Z -1.3333, A 0.000, B 0.000, C 0.000 }
gfCNCPoint1[11648] = {X 227.1564, Y 46.7702, Z -1.3333, A 0.000, B 0.000, C 0.000 }
gfCNCPoint1[11649] = {X 226.6704, Y 47.5438, Z -1.3333, A 0.000, B 0.000, C 0.000 }
gfCNCPoint1[11650] = {X 226.0243, Y 48.1899, Z -1.3333, A 0.000, B 0.000, C 0.000 }
gfCNCPoint1[11651] = {X 225.2507, Y 48.6760, Z -1.3333, A 0.000, B 0.000, C 0.000 }
gfCNCPoint1[11652] = {X 224.3884, Y 48.9777, Z -1.3333, A 0.000, B 0.000, C 0.000 }
gfCNCPoint1[11653] = {X 223.4805, Y 49.0800, Z -1.3333, A 0.000, B 0.000, C 0.000 }
gfCNCPoint1[11654] = {X 217.0370, Y 49.0800, Z -1.3333, A 0.000, B 0.000, C 0.000 }
gfCNCPoint1[11655] = {X 216.1337, Y 48.9787, Z -1.3333, A 0.000, B 0.000, C 0.000 }
gfCNCPoint1[11656] = {X 215.2752, Y 48.6800, Z -1.3333, A 0.000, B 0.000, C 0.000 }
gfCNCPoint1[11657] = {X 214.5041, Y 48.1986, Z -1.3333, A 0.000, B 0.000, C 0.000 }
gfCNCPoint1[11658] = {X 213.8588, Y 47.5584, Z -1.3333, A 0.000, B 0.000, C 0.000 }
gfCNCPoint1[11659] = {X 213.3712, Y 46.7912, Z -1.3333, A 0.000, B 0.000, C 0.000 }
gfCNCPoint1[11660] = {X 213.0656, Y 45.9351, Z -1.3333, A 0.000, B 0.000, C 0.000 }
gfCNCPoint1[11661] = {X 212.9571, Y 45.0325, Z -1.3333, A 0.000, B 0.000, C 0.000 }
gfCNCPoint1[11662] = {X 212.9570, Y 44.2008, Z -1.3333, A 0.000, B 0.000, C 0.000 }
gfCNCPoint1[11663] = {X 213.0250, Y 43.4649, Z -1.3333, A 0.000, B 0.000, C 0.000 }
gfCNCPoint1[11664] = {X 213.2265, Y 42.7538, Z -1.3333, A 0.000, B 0.000, C 0.000 }
gfCNCPoint1[11665] = {X 213.5548, Y 42.0917, Z -1.3333, A 0.000, B 0.000, C 0.000 }
gfCNCPoint1[11666] = {X 213.9987, Y 41.5008, Z -1.3333, A 0.000, B 0.000, C 0.000 }
gfCNCPoint1[11667] = {X 214.4811, Y 40.9687, Z -1.3333, A 0.000, B 0.000, C 0.000 }
gfCNCPoint1[11668] = {X 214.4862, Y 40.3072, Z -1.3333, A 0.000, B 0.000, C 0.000 }
gfCNCPoint1[11669] = {X 214.4862, Y 28.5743, Z -1.3333, A 0.000, B 0.000, C 0.000 }
gfCNCPoint1[11670] = {X 210.4862, Y 28.5743, Z -1.3333, A 0.000, B 0.000, C 0.000 }
gfCNCPoint1[11671] = {X 214.5662, Y 28.5743, Z -1.3333, A 0.000, B 0.000, C 0.000 }
gfCNCPoint1[11672] = {X 214.5662, Y 17.4611, Z -1.3333, A 0.000, B 0.000, C 0.000 }
gfCNCPoint1[11673] = {X 214.5609, Y 16.7687, Z -1.3333, A 0.000, B 0.000, C 0.000 }
gfCNCPoint1[11674] = {X 214.5601, Y 16.1861, Z -1.3333, A 0.000, B 0.000, C 0.000 }
gfCNCPoint1[11675] = {X 214.5756, Y 16.1310, Z -1.3333, A 0.000, B 0.000, C 0.000 }
gfCNCPoint1[11676] = {X 214.4979, Y 16.0688, Z -1.3333, A 0.000, B 0.000, C 0.000 }
gfCNCPoint1[11677] = {X 214.4218, Y 16.0047, Z -1.3333, A 0.000, B 0.000, C 0.000 }
gfCNCPoint1[11678] = {X 213.8374, Y 15.3785, Z -1.3333, A 0.000, B 0.000, C 0.000 }
gfCNCPoint1[11679] = {X 213.3996, Y 14.6422, Z -1.3333, A 0.000, B 0.000, C 0.000 }
gfCNCPoint1[11680] = {X 213.1287, Y 13.8296, Z -1.3333, A 0.000, B 0.000, C 0.000 }
gfCNCPoint1[11681] = {X 213.0370, Y 12.9779, Z -1.3333, A 0.000, B 0.000, C 0.000 }
gfCNCPoint1[11682] = {X 213.0370, Y 12.1868, Z -1.3333, A 0.000, B 0.000, C 0.000 }
gfCNCPoint1[11683] = {X 213.1373, Y 11.2967, Z -1.3333, A 0.000, B 0.000, C 0.000 }
gfCNCPoint1[11684] = {X 213.4331, Y 10.4513, Z -1.3333, A 0.000, B 0.000, C 0.000 }
gfCNCPoint1[11685] = {X 213.9097, Y 9.6929, Z -1.3333, A 0.000, B 0.000, C 0.000 }
gfCNCPoint1[11686] = {X 214.5431, Y 9.0595, Z -1.3333, A 0.000, B 0.000, C 0.000 }
gfCNCPoint1[11687] = {X 215.3015, Y 8.5829, Z -1.3333, A 0.000, B 0.000, C 0.000 }
gfCNCPoint1[11688] = {X 216.1469, Y 8.2871, Z -1.3333, A 0.000, B 0.000, C 0.000 }
gfCNCPoint1[11689] = {X 217.0370, Y 8.1868, Z -1.3333, A 0.000, B 0.000, C 0.000 }
gfCNCPoint1[11690] = {X 223.4805, Y 8.1868, Z -1.3333, A 0.000, B 0.000, C 0.000 }
gfCNCPoint1[11691] = {X 224.3706, Y 8.2871, Z -1.3333, A 0.000, B 0.000, C 0.000 }
gfCNCPoint1[11692] = {X 225.2160, Y 8.5829, Z -1.3333, A 0.000, B 0.000, C 0.000 }
gfCNCPoint1[11693] = {X 225.9744, Y 9.0595, Z -1.3333, A 0.000, B 0.000, C 0.000 }
gfCNCPoint1[11694] = {X 226.6078, Y 9.6929, Z -1.3333, A 0.000, B 0.000, C 0.000 }
gfCNCPoint1[11695] = {X 227.0844, Y 10.4513, Z -1.3333, A 0.000, B 0.000, C 0.000 }
gfCNCPoint1[11696] = {X 227.3802, Y 11.2967, Z -1.3333, A 0.000, B 0.000, C 0.000 }
gfCNCPoint1[11697] = {X 227.4805, Y 12.1868, Z -1.3333, A 0.000, B 0.000, C 0.000 }
gfCNCPoint1[11698] = {X 227.4803, Y 13.0192, Z -1.3333, A 0.000, B 0.000, C 0.000 }
gfCNCPoint1[11699] = {X 227.3716, Y 13.9051, Z -1.3333, A 0.000, B 0.000, C 0.000 }
gfCNCPoint1[11700] = {X 227.0691, Y 14.7449, Z -1.3333, A 0.000, B 0.000, C 0.000 }
gfCNCPoint1[11701] = {X 226.5879, Y 15.4967, Z -1.3333, A 0.000, B 0.000, C 0.000 }
gfCNCPoint1[11702] = {X 225.9520, Y 16.1231, Z -1.3333, A 0.000, B 0.000, C 0.000 }
gfCNCPoint1[11703] = {X 225.9529, Y 41.0669, Z -1.3333, A 0.000, B 0.000, C 0.000 }
gfCNCPoint1[11704] = {X 226.0918, Y 41.1788, Z -1.3333, A 0.000, B 0.000, C 0.000 }
gfCNCPoint1[11705] = {X 226.6778, Y 41.8053, Z -1.3333, A 0.000, B 0.000, C 0.000 }
gfCNCPoint1[11706] = {X 227.1168, Y 42.5423, Z -1.3333, A 0.000, B 0.000, C 0.000 }
gfCNCPoint1[11707] = {X 227.3885, Y 43.3560, Z -1.3333, A 0.000, B 0.000, C 0.000 }
gfCNCPoint1[11708] = {X 227.4805, Y 44.2089, Z -1.3333, A 0.000, B 0.000, C 0.000 }
gfCNCPoint1[11709] = {X 227.4805, Y 45.0000, Z -1.3333, A 0.000, B 0.000, C 0.000 }
gfCNCPoint1[11710] = {X 227.3802, Y 45.8901, Z -1.3333, A 0.000, B 0.000, C 0.000 }
gfCNCPoint1[11711] = {X 227.0844, Y 46.7355, Z -1.3333, A 0.000, B 0.000, C 0.000 }
gfCNCPoint1[11712] = {X 226.6078, Y 47.4940, Z -1.3333, A 0.000, B 0.000, C 0.000 }
gfCNCPoint1[11713] = {X 225.9744, Y 48.1273, Z -1.3333, A 0.000, B 0.000, C 0.000 }
gfCNCPoint1[11714] = {X 225.2160, Y 48.6039, Z -1.3333, A 0.000, B 0.000, C 0.000 }
gfCNCPoint1[11715] = {X 224.3706, Y 48.8997, Z -1.3333, A 0.000, B 0.000, C 0.000 }
gfCNCPoint1[11716] = {X 223.4805, Y 49.0000, Z -1.3333, A 0.000, B 0.000, C 0.000 }
gfCNCPoint1[11717] = {X 217.0370, Y 49.0000, Z -1.3333, A 0.000, B 0.000, C 0.000 }
gfCNCPoint1[11718] = {X 216.1469, Y 48.8997, Z -1.3333, A 0.000, B 0.000, C 0.000 }
gfCNCPoint1[11719] = {X 215.3015, Y 48.6039, Z -1.3333, A 0.000, B 0.000, C 0.000 }
gfCNCPoint1[11720] = {X 214.5430, Y 48.1273, Z -1.3333, A 0.000, B 0.000, C 0.000 }
gfCNCPoint1[11721] = {X 213.9097, Y 47.4939, Z -1.3333, A 0.000, B 0.000, C 0.000 }
gfCNCPoint1[11722] = {X 213.4331, Y 46.7355, Z -1.3333, A 0.000, B 0.000, C 0.000 }
gfCNCPoint1[11723] = {X 213.1373, Y 45.8900, Z -1.3333, A 0.000, B 0.000, C 0.000 }
gfCNCPoint1[11724] = {X 213.0370, Y 45.0000, Z -1.3333, A 0.000, B 0.000, C 0.000 }
gfCNCPoint1[11725] = {X 213.0370, Y 44.2008, Z -1.3333, A 0.000, B 0.000, C 0.000 }
gfCNCPoint1[11726] = {X 213.1551, Y 43.2433, Z -1.3333, A 0.000, B 0.000, C 0.000 }
gfCNCPoint1[11727] = {X 213.5024, Y 42.3433, Z -1.3333, A 0.000, B 0.000, C 0.000 }
gfCNCPoint1[11728] = {X 214.0580, Y 41.5546, Z -1.3333, A 0.000, B 0.000, C 0.000 }
gfCNCPoint1[11729] = {X 214.5609, Y 40.9999, Z -1.3333, A 0.000, B 0.000, C 0.000 }
gfCNCPoint1[11730] = {X 214.5662, Y 40.3075, Z -1.3333, A 0.000, B 0.000, C 0.000 }
gfCNCPoint1[11731] = {X 214.5662, Y 28.5743, Z -1.3333, A 0.000, B 0.000, C 0.000 }
gfCNCPoint1[11732] = {X 210.4862, Y 28.5743, Z -1.3333, A 0.000, B 0.000, C 0.000 }
gfCNCPoint1[11733] = {X 210.4862, Y 28.5743, Z 1.6667, A 0.000, B 0.000, C 0.000 }
gfCNCPoint1[11734] = {X 210.4862, Y 28.5743, Z 11.0000, A 0.000, B 0.000, C 0.000 }
gfCNCPoint1[11735] = {X 273.6027, Y 28.5937, Z 11.0000, A 0.000, B 0.000, C 0.000 }
gfCNCPoint1[11736] = {X 273.6027, Y 28.5937, Z 1.6667, A 0.000, B 0.000, C 0.000 }
gfCNCPoint1[11737] = {X 273.6027, Y 28.5937, Z -1.3333, A 0.000, B 0.000, C 0.000 }
gfCNCPoint1[11738] = {X 269.5227, Y 28.5937, Z -1.3333, A 0.000, B 0.000, C 0.000 }
gfCNCPoint1[11739] = {X 269.5226, Y 40.9126, Z -1.3333, A 0.000, B 0.000, C 0.000 }
gfCNCPoint1[11740] = {X 269.5366, Y 40.9238, Z -1.3333, A 0.000, B 0.000, C 0.000 }
gfCNCPoint1[11741] = {X 270.1693, Y 41.5934, Z -1.3333, A 0.000, B 0.000, C 0.000 }
gfCNCPoint1[11742] = {X 270.6457, Y 42.3819, Z -1.3333, A 0.000, B 0.000, C 0.000 }
gfCNCPoint1[11743] = {X 270.9441, Y 43.2535, Z -1.3333, A 0.000, B 0.000, C 0.000 }
gfCNCPoint1[11744] = {X 271.0508, Y 44.1686, Z -1.3333, A 0.000, B 0.000, C 0.000 }
gfCNCPoint1[11745] = {X 271.0510, Y 45.0000, Z -1.3333, A 0.000, B 0.000, C 0.000 }
gfCNCPoint1[11746] = {X 270.9427, Y 45.9613, Z -1.3333, A 0.000, B 0.000, C 0.000 }
gfCNCPoint1[11747] = {X 270.6232, Y 46.8744, Z -1.3333, A 0.000, B 0.000, C 0.000 }
gfCNCPoint1[11748] = {X 270.1085, Y 47.6935, Z -1.3333, A 0.000, B 0.000, C 0.000 }
gfCNCPoint1[11749] = {X 269.4245, Y 48.3775, Z -1.3333, A 0.000, B 0.000, C 0.000 }
gfCNCPoint1[11750] = {X 268.6054, Y 48.8922, Z -1.3333, A 0.000, B 0.000, C 0.000 }
gfCNCPoint1[11751] = {X 267.6923, Y 49.2117, Z -1.3333, A 0.000, B 0.000, C 0.000 }
gfCNCPoint1[11752] = {X 266.7310, Y 49.3200, Z -1.3333, A 0.000, B 0.000, C 0.000 }
gfCNCPoint1[11753] = {X 260.2876, Y 49.3200, Z -1.3333, A 0.000, B 0.000, C 0.000 }
gfCNCPoint1[11754] = {X 259.3310, Y 49.2128, Z -1.3333, A 0.000, B 0.000, C 0.000 }
gfCNCPoint1[11755] = {X 258.4219, Y 48.8963, Z -1.3333, A 0.000, B 0.000, C 0.000 }
gfCNCPoint1[11756] = {X 257.6054, Y 48.3865, Z -1.3333, A 0.000, B 0.000, C 0.000 }
gfCNCPoint1[11757] = {X 256.9221, Y 47.7085, Z -1.3333, A 0.000, B 0.000, C 0.000 }
gfCNCPoint1[11758] = {X 256.4059, Y 46.8960, Z -1.3333, A 0.000, B 0.000, C 0.000 }
gfCNCPoint1[11759] = {X 256.0824, Y 45.9894, Z -1.3333, A 0.000, B 0.000, C 0.000 }
gfCNCPoint1[11760] = {X 255.9677, Y 45.0336, Z -1.3333, A 0.000, B 0.000, C 0.000 }
gfCNCPoint1[11761] = {X 255.9680, Y 44.1494, Z -1.3333, A 0.000, B 0.000, C 0.000 }
gfCNCPoint1[11762] = {X 256.0784, Y 43.2364, Z -1.3333, A 0.000, B 0.000, C 0.000 }
gfCNCPoint1[11763] = {X 256.3796, Y 42.3675, Z -1.3333, A 0.000, B 0.000, C 0.000 }
gfCNCPoint1[11764] = {X 256.8579, Y 41.5821, Z -1.3333, A 0.000, B 0.000, C 0.000 }
gfCNCPoint1[11765] = {X 257.4915, Y 40.9157, Z -1.3333, A 0.000, B 0.000, C 0.000 }
gfCNCPoint1[11766] = {X 257.4915, Y 34.4738, Z -1.3333, A 0.000, B 0.000, C 0.000 }
gfCNCPoint1[11767] = {X 254.7664, Y 34.4738, Z -1.3333, A 0.000, B 0.000, C 0.000 }
gfCNCPoint1[11768] = {X 250.4835, Y 42.8178, Z -1.3333, A 0.000, B 0.000, C 0.000 }
gfCNCPoint1[11769] = {X 250.6526, Y 43.4859, Z -1.3333, A 0.000, B 0.000, C 0.000 }
gfCNCPoint1[11770] = {X 250.7134, Y 44.1723, Z -1.3333, A 0.000, B 0.000, C 0.000 }
gfCNCPoint1[11771] = {X 250.7136, Y 45.0000, Z -1.3333, A 0.000, B 0.000, C 0.000 }
gfCNCPoint1[11772] = {X 250.6052, Y 45.9613, Z -1.3333, A 0.000, B 0.000, C 0.000 }
gfCNCPoint1[11773] = {X 250.2857, Y 46.8744, Z -1.3333, A 0.000, B 0.000, C 0.000 }
gfCNCPoint1[11774] = {X 249.7711, Y 47.6935, Z -1.3333, A 0.000, B 0.000, C 0.000 }
gfCNCPoint1[11775] = {X 249.0870, Y 48.3775, Z -1.3333, A 0.000, B 0.000, C 0.000 }
gfCNCPoint1[11776] = {X 248.2679, Y 48.8922, Z -1.3333, A 0.000, B 0.000, C 0.000 }
gfCNCPoint1[11777] = {X 247.3548, Y 49.2117, Z -1.3333, A 0.000, B 0.000, C 0.000 }
gfCNCPoint1[11778] = {X 246.3936, Y 49.3200, Z -1.3333, A 0.000, B 0.000, C 0.000 }
gfCNCPoint1[11779] = {X 239.8075, Y 49.3200, Z -1.3333, A 0.000, B 0.000, C 0.000 }
gfCNCPoint1[11780] = {X 238.8462, Y 49.2117, Z -1.3333, A 0.000, B 0.000, C 0.000 }
gfCNCPoint1[11781] = {X 237.9331, Y 48.8922, Z -1.3333, A 0.000, B 0.000, C 0.000 }
gfCNCPoint1[11782] = {X 237.1141, Y 48.3775, Z -1.3333, A 0.000, B 0.000, C 0.000 }
gfCNCPoint1[11783] = {X 236.4300, Y 47.6935, Z -1.3333, A 0.000, B 0.000, C 0.000 }
gfCNCPoint1[11784] = {X 235.9153, Y 46.8745, Z -1.3333, A 0.000, B 0.000, C 0.000 }
gfCNCPoint1[11785] = {X 235.5958, Y 45.9614, Z -1.3333, A 0.000, B 0.000, C 0.000 }
gfCNCPoint1[11786] = {X 235.4875, Y 45.0001, Z -1.3333, A 0.000, B 0.000, C 0.000 }
gfCNCPoint1[11787] = {X 235.4879, Y 44.1494, Z -1.3333, A 0.000, B 0.000, C 0.000 }
gfCNCPoint1[11788] = {X 235.5856, Y 43.2935, Z -1.3333, A 0.000, B 0.000, C 0.000 }
gfCNCPoint1[11789] = {X 235.8511, Y 42.4740, Z -1.3333, A 0.000, B 0.000, C 0.000 }
gfCNCPoint1[11790] = {X 236.2739, Y 41.7236, Z -1.3333, A 0.000, B 0.000, C 0.000 }
gfCNCPoint1[11791] = {X 236.8373, Y 41.0719, Z -1.3333, A 0.000, B 0.000, C 0.000 }
gfCNCPoint1[11792] = {X 237.5187, Y 40.5449, Z -1.3333, A 0.000, B 0.000, C 0.000 }
gfCNCPoint1[11793] = {X 238.2911, Y 40.1637, Z -1.3333, A 0.000, B 0.000, C 0.000 }
gfCNCPoint1[11794] = {X 242.2808, Y 32.3544, Z -1.3333, A 0.000, B 0.000, C 0.000 }
gfCNCPoint1[11795] = {X 241.1109, Y 31.5681, Z -1.3333, A 0.000, B 0.000, C 0.000 }
gfCNCPoint1[11796] = {X 240.0479, Y 30.6425, Z -1.3333, A 0.000, B 0.000, C 0.000 }
gfCNCPoint1[11797] = {X 239.1082, Y 29.5919, Z -1.3333, A 0.000, B 0.000, C 0.000 }
gfCNCPoint1[11798] = {X 238.3064, Y 28.4326, Z -1.3333, A 0.000, B 0.000, C 0.000 }
gfCNCPoint1[11799] = {X 237.6550, Y 27.1827, Z -1.3333, A 0.000, B 0.000, C 0.000 }
gfCNCPoint1[11800] = {X 237.1639, Y 25.8615, Z -1.3333, A 0.000, B 0.000, C 0.000 }
gfCNCPoint1[11801] = {X 236.7438, Y 24.0500, Z -1.3333, A 0.000, B 0.000, C 0.000 }
gfCNCPoint1[11802] = {X 236.5296, Y 22.2028, Z -1.3333, A 0.000, B 0.000, C 0.000 }
gfCNCPoint1[11803] = {X 236.5243, Y 20.3433, Z -1.3333, A 0.000, B 0.000, C 0.000 }
gfCNCPoint1[11804] = {X 236.7277, Y 18.4949, Z -1.3333, A 0.000, B 0.000, C 0.000 }
gfCNCPoint1[11805] = {X 237.1375, Y 16.6811, Z -1.3333, A 0.000, B 0.000, C 0.000 }
gfCNCPoint1[11806] = {X 237.7077, Y 15.1056, Z -1.3333, A 0.000, B 0.000, C 0.000 }
gfCNCPoint1[11807] = {X 238.4945, Y 13.6262, Z -1.3333, A 0.000, B 0.000, C 0.000 }
gfCNCPoint1[11808] = {X 239.4822, Y 12.2728, Z -1.3333, A 0.000, B 0.000, C 0.000 }
gfCNCPoint1[11809] = {X 240.6510, Y 11.0722, Z -1.3333, A 0.000, B 0.000, C 0.000 }
gfCNCPoint1[11810] = {X 241.9775, Y 10.0485, Z -1.3333, A 0.000, B 0.000, C 0.000 }
gfCNCPoint1[11811] = {X 243.4351, Y 9.2223, Z -1.3333, A 0.000, B 0.000, C 0.000 }
gfCNCPoint1[11812] = {X 244.9948, Y 8.6100, Z -1.3333, A 0.000, B 0.000, C 0.000 }
gfCNCPoint1[11813] = {X 246.6252, Y 8.2239, Z -1.3333, A 0.000, B 0.000, C 0.000 }
gfCNCPoint1[11814] = {X 248.7221, Y 7.9524, Z -1.3333, A 0.000, B 0.000, C 0.000 }
gfCNCPoint1[11815] = {X 250.8349, Y 7.8719, Z -1.3333, A 0.000, B 0.000, C 0.000 }
gfCNCPoint1[11816] = {X 266.7634, Y 7.8719, Z -1.3333, A 0.000, B 0.000, C 0.000 }
gfCNCPoint1[11817] = {X 267.7183, Y 7.9867, Z -1.3333, A 0.000, B 0.000, C 0.000 }
gfCNCPoint1[11818] = {X 268.6243, Y 8.3098, Z -1.3333, A 0.000, B 0.000, C 0.000 }
gfCNCPoint1[11819] = {X 269.4364, Y 8.8252, Z -1.3333, A 0.000, B 0.000, C 0.000 }
gfCNCPoint1[11820] = {X 270.1144, Y 9.5074, Z -1.3333, A 0.000, B 0.000, C 0.000 }
gfCNCPoint1[11821] = {X 270.6247, Y 10.3227, Z -1.3333, A 0.000, B 0.000, C 0.000 }
gfCNCPoint1[11822] = {X 270.9422, Y 11.2306, Z -1.3333, A 0.000, B 0.000, C 0.000 }
gfCNCPoint1[11823] = {X 271.0510, Y 12.1863, Z -1.3333, A 0.000, B 0.000, C 0.000 }
gfCNCPoint1[11824] = {X 271.0508, Y 13.0225, Z -1.3333, A 0.000, B 0.000, C 0.000 }
gfCNCPoint1[11825] = {X 270.9424, Y 13.9408, Z -1.3333, A 0.000, B 0.000, C 0.000 }
gfCNCPoint1[11826] = {X 270.6410, Y 14.8150, Z -1.3333, A 0.000, B 0.000, C 0.000 }
gfCNCPoint1[11827] = {X 270.1605, Y 15.6050, Z -1.3333, A 0.000, B 0.000, C 0.000 }
gfCNCPoint1[11828] = {X 269.5228, Y 16.2747, Z -1.3333, A 0.000, B 0.000, C 0.000 }
gfCNCPoint1[11829] = {X 269.5227, Y 28.5937, Z -1.3333, A 0.000, B 0.000, C 0.000 }
gfCNCPoint1[11830] = {X 273.5227, Y 28.5937, Z -1.3333, A 0.000, B 0.000, C 0.000 }
gfCNCPoint1[11831] = {X 269.4427, Y 28.5937, Z -1.3333, A 0.000, B 0.000, C 0.000 }
gfCNCPoint1[11832] = {X 269.4426, Y 40.9510, Z -1.3333, A 0.000, B 0.000, C 0.000 }
gfCNCPoint1[11833] = {X 269.4856, Y 40.9854, Z -1.3333, A 0.000, B 0.000, C 0.000 }
gfCNCPoint1[11834] = {X 270.1062, Y 41.6425, Z -1.3333, A 0.000, B 0.000, C 0.000 }
gfCNCPoint1[11835] = {X 270.5735, Y 42.4163, Z -1.3333, A 0.000, B 0.000, C 0.000 }
gfCNCPoint1[11836] = {X 270.8661, Y 43.2715, Z -1.3333, A 0.000, B 0.000, C 0.000 }
gfCNCPoint1[11837] = {X 270.9708, Y 44.1693, Z -1.3333, A 0.000, B 0.000, C 0.000 }
gfCNCPoint1[11838] = {X 270.9710, Y 45.0000, Z -1.3333, A 0.000, B 0.000, C 0.000 }
gfCNCPoint1[11839] = {X 270.8647, Y 45.9435, Z -1.3333, A 0.000, B 0.000, C 0.000 }
gfCNCPoint1[11840] = {X 270.5511, Y 46.8397, Z -1.3333, A 0.000, B 0.000, C 0.000 }
gfCNCPoint1[11841] = {X 270.0460, Y 47.6436, Z -1.3333, A 0.000, B 0.000, C 0.000 }
gfCNCPoint1[11842] = {X 269.3746, Y 48.3150, Z -1.3333, A 0.000, B 0.000, C 0.000 }
gfCNCPoint1[11843] = {X 268.5707, Y 48.8201, Z -1.3333, A 0.000, B 0.000, C 0.000 }
gfCNCPoint1[11844] = {X 267.6745, Y 49.1337, Z -1.3333, A 0.000, B 0.000, C 0.000 }
gfCNCPoint1[11845] = {X 266.7310, Y 49.2400, Z -1.3333, A 0.000, B 0.000, C 0.000 }
gfCNCPoint1[11846] = {X 260.2876, Y 49.2400, Z -1.3333, A 0.000, B 0.000, C 0.000 }
gfCNCPoint1[11847] = {X 259.3487, Y 49.1347, Z -1.3333, A 0.000, B 0.000, C 0.000 }
gfCNCPoint1[11848] = {X 258.4564, Y 48.8242, Z -1.3333, A 0.000, B 0.000, C 0.000 }
gfCNCPoint1[11849] = {X 257.6550, Y 48.3238, Z -1.3333, A 0.000, B 0.000, C 0.000 }
gfCNCPoint1[11850] = {X 256.9844, Y 47.6583, Z -1.3333, A 0.000, B 0.000, C 0.000 }
gfCNCPoint1[11851] = {X 256.4777, Y 46.8609, Z -1.3333, A 0.000, B 0.000, C 0.000 }
gfCNCPoint1[11852] = {X 256.1603, Y 45.9711, Z -1.3333, A 0.000, B 0.000, C 0.000 }
gfCNCPoint1[11853] = {X 256.0477, Y 45.0330, Z -1.3333, A 0.000, B 0.000, C 0.000 }
gfCNCPoint1[11854] = {X 256.0480, Y 44.1505, Z -1.3333, A 0.000, B 0.000, C 0.000 }
gfCNCPoint1[11855] = {X 256.1585, Y 43.2454, Z -1.3333, A 0.000, B 0.000, C 0.000 }
gfCNCPoint1[11856] = {X 256.4599, Y 42.3850, Z -1.3333, A 0.000, B 0.000, C 0.000 }
gfCNCPoint1[11857] = {X 256.9383, Y 41.6088, Z -1.3333, A 0.000, B 0.000, C 0.000 }
gfCNCPoint1[11858] = {X 257.5715, Y 40.9529, Z -1.3333, A 0.000, B 0.000, C 0.000 }
gfCNCPoint1[11859] = {X 257.5715, Y 34.3938, Z -1.3333, A 0.000, B 0.000, C 0.000 }
gfCNCPoint1[11860] = {X 254.7176, Y 34.3938, Z -1.3333, A 0.000, B 0.000, C 0.000 }
gfCNCPoint1[11861] = {X 250.3968, Y 42.8116, Z -1.3333, A 0.000, B 0.000, C 0.000 }
gfCNCPoint1[11862] = {X 250.5709, Y 43.4826, Z -1.3333, A 0.000, B 0.000, C 0.000 }
gfCNCPoint1[11863] = {X 250.6334, Y 44.1730, Z -1.3333, A 0.000, B 0.000, C 0.000 }
gfCNCPoint1[11864] = {X 250.6336, Y 45.0000, Z -1.3333, A 0.000, B 0.000, C 0.000 }
gfCNCPoint1[11865] = {X 250.5273, Y 45.9435, Z -1.3333, A 0.000, B 0.000, C 0.000 }
gfCNCPoint1[11866] = {X 250.2137, Y 46.8397, Z -1.3333, A 0.000, B 0.000, C 0.000 }
gfCNCPoint1[11867] = {X 249.7085, Y 47.6436, Z -1.3333, A 0.000, B 0.000, C 0.000 }
gfCNCPoint1[11868] = {X 249.0372, Y 48.3150, Z -1.3333, A 0.000, B 0.000, C 0.000 }
gfCNCPoint1[11869] = {X 248.2332, Y 48.8201, Z -1.3333, A 0.000, B 0.000, C 0.000 }
gfCNCPoint1[11870] = {X 247.3370, Y 49.1337, Z -1.3333, A 0.000, B 0.000, C 0.000 }
gfCNCPoint1[11871] = {X 246.3936, Y 49.2400, Z -1.3333, A 0.000, B 0.000, C 0.000 }
gfCNCPoint1[11872] = {X 239.8075, Y 49.2400, Z -1.3333, A 0.000, B 0.000, C 0.000 }
gfCNCPoint1[11873] = {X 238.8640, Y 49.1337, Z -1.3333, A 0.000, B 0.000, C 0.000 }
gfCNCPoint1[11874] = {X 237.9679, Y 48.8201, Z -1.3333, A 0.000, B 0.000, C 0.000 }
gfCNCPoint1[11875] = {X 237.1639, Y 48.3150, Z -1.3333, A 0.000, B 0.000, C 0.000 }
gfCNCPoint1[11876] = {X 236.4926, Y 47.6436, Z -1.3333, A 0.000, B 0.000, C 0.000 }
gfCNCPoint1[11877] = {X 235.9874, Y 46.8397, Z -1.3333, A 0.000, B 0.000, C 0.000 }
gfCNCPoint1[11878] = {X 235.6738, Y 45.9436, Z -1.3333, A 0.000, B 0.000, C 0.000 }
gfCNCPoint1[11879] = {X 235.5675, Y 45.0001, Z -1.3333, A 0.000, B 0.000, C 0.000 }
gfCNCPoint1[11880] = {X 235.5679, Y 44.1505, Z -1.3333, A 0.000, B 0.000, C 0.000 }
gfCNCPoint1[11881] = {X 235.6649, Y 43.3054, Z -1.3333, A 0.000, B 0.000, C 0.000 }
gfCNCPoint1[11882] = {X 235.9285, Y 42.4967, Z -1.3333, A 0.000, B 0.000, C 0.000 }
gfCNCPoint1[11883] = {X 236.3483, Y 41.7570, Z -1.3333, A 0.000, B 0.000, C 0.000 }
gfCNCPoint1[11884] = {X 236.9073, Y 41.1159, Z -1.3333, A 0.000, B 0.000, C 0.000 }
gfCNCPoint1[11885] = {X 237.5830, Y 40.5992, Z -1.3333, A 0.000, B 0.000, C 0.000 }
gfCNCPoint1[11886] = {X 238.3482, Y 40.2278, Z -1.3333, A 0.000, B 0.000, C 0.000 }
gfCNCPoint1[11887] = {X 242.3865, Y 32.3233, Z -1.3333, A 0.000, B 0.000, C 0.000 }
gfCNCPoint1[11888] = {X 241.2097, Y 31.5428, Z -1.3333, A 0.000, B 0.000, C 0.000 }
gfCNCPoint1[11889] = {X 240.1400, Y 30.6208, Z -1.3333, A 0.000, B 0.000, C 0.000 }
gfCNCPoint1[11890] = {X 239.1945, Y 29.5720, Z -1.3333, A 0.000, B 0.000, C 0.000 }
gfCNCPoint1[11891] = {X 238.3880, Y 28.4129, Z -1.3333, A 0.000, B 0.000, C 0.000 }
gfCNCPoint1[11892] = {X 237.7332, Y 27.1617, Z -1.3333, A 0.000, B 0.000, C 0.000 }
gfCNCPoint1[11893] = {X 237.2405, Y 25.8383, Z -1.3333, A 0.000, B 0.000, C 0.000 }
gfCNCPoint1[11894] = {X 236.8225, Y 24.0357, Z -1.3333, A 0.000, B 0.000, C 0.000 }
gfCNCPoint1[11895] = {X 236.6095, Y 22.1976, Z -1.3333, A 0.000, B 0.000, C 0.000 }
gfCNCPoint1[11896] = {X 236.6042, Y 20.3472, Z -1.3333, A 0.000, B 0.000, C 0.000 }
gfCNCPoint1[11897] = {X 236.8067, Y 18.5079, Z -1.3333, A 0.000, B 0.000, C 0.000 }
gfCNCPoint1[11898] = {X 237.2144, Y 16.7029, Z -1.3333, A 0.000, B 0.000, C 0.000 }
gfCNCPoint1[11899] = {X 237.7808, Y 15.1380, Z -1.3333, A 0.000, B 0.000, C 0.000 }
gfCNCPoint1[11900] = {X 238.5624, Y 13.6686, Z -1.3333, A 0.000, B 0.000, C 0.000 }
gfCNCPoint1[11901] = {X 239.5434, Y 12.3242, Z -1.3333, A 0.000, B 0.000, C 0.000 }
gfCNCPoint1[11902] = {X 240.7044, Y 11.1317, Z -1.3333, A 0.000, B 0.000, C 0.000 }
gfCNCPoint1[11903] = {X 242.0220, Y 10.1150, Z -1.3333, A 0.000, B 0.000, C 0.000 }
gfCNCPoint1[11904] = {X 243.4699, Y 9.2943, Z -1.3333, A 0.000, B 0.000, C 0.000 }
gfCNCPoint1[11905] = {X 245.0191, Y 8.6862, Z -1.3333, A 0.000, B 0.000, C 0.000 }
gfCNCPoint1[11906] = {X 246.6386, Y 8.3028, Z -1.3333, A 0.000, B 0.000, C 0.000 }
gfCNCPoint1[11907] = {X 248.7286, Y 8.0321, Z -1.3333, A 0.000, B 0.000, C 0.000 }
gfCNCPoint1[11908] = {X 250.8346, Y 7.9519, Z -1.3333, A 0.000, B 0.000, C 0.000 }
gfCNCPoint1[11909] = {X 266.7627, Y 7.9519, Z -1.3333, A 0.000, B 0.000, C 0.000 }
gfCNCPoint1[11910] = {X 267.7000, Y 8.0645, Z -1.3333, A 0.000, B 0.000, C 0.000 }
gfCNCPoint1[11911] = {X 268.5892, Y 8.3817, Z -1.3333, A 0.000, B 0.000, C 0.000 }
gfCNCPoint1[11912] = {X 269.3863, Y 8.8875, Z -1.3333, A 0.000, B 0.000, C 0.000 }
gfCNCPoint1[11913] = {X 270.0517, Y 9.5571, Z -1.3333, A 0.000, B 0.000, C 0.000 }
gfCNCPoint1[11914] = {X 270.5526, Y 10.3573, Z -1.3333, A 0.000, B 0.000, C 0.000 }
gfCNCPoint1[11915] = {X 270.8642, Y 11.2485, Z -1.3333, A 0.000, B 0.000, C 0.000 }
gfCNCPoint1[11916] = {X 270.9710, Y 12.1864, Z -1.3333, A 0.000, B 0.000, C 0.000 }
gfCNCPoint1[11917] = {X 270.9708, Y 13.0217, Z -1.3333, A 0.000, B 0.000, C 0.000 }
gfCNCPoint1[11918] = {X 270.8623, Y 13.9320, Z -1.3333, A 0.000, B 0.000, C 0.000 }
gfCNCPoint1[11919] = {X 270.5607, Y 14.7977, Z -1.3333, A 0.000, B 0.000, C 0.000 }
gfCNCPoint1[11920] = {X 270.0801, Y 15.5783, Z -1.3333, A 0.000, B 0.000, C 0.000 }
gfCNCPoint1[11921] = {X 269.4428, Y 16.2374, Z -1.3333, A 0.000, B 0.000, C 0.000 }
gfCNCPoint1[11922] = {X 269.4427, Y 28.5937, Z -1.3333, A 0.000, B 0.000, C 0.000 }
gfCNCPoint1[11923] = {X 273.4427, Y 28.5937, Z -1.3333, A 0.000, B 0.000, C 0.000 }
gfCNCPoint1[11924] = {X 269.3627, Y 28.5937, Z -1.3333, A 0.000, B 0.000, C 0.000 }
gfCNCPoint1[11925] = {X 269.3626, Y 40.9895, Z -1.3333, A 0.000, B 0.000, C 0.000 }
gfCNCPoint1[11926] = {X 269.4346, Y 41.0471, Z -1.3333, A 0.000, B 0.000, C 0.000 }
gfCNCPoint1[11927] = {X 270.0431, Y 41.6917, Z -1.3333, A 0.000, B 0.000, C 0.000 }
gfCNCPoint1[11928] = {X 270.5013, Y 42.4507, Z -1.3333, A 0.000, B 0.000, C 0.000 }
gfCNCPoint1[11929] = {X 270.7882, Y 43.2895, Z -1.3333, A 0.000, B 0.000, C 0.000 }
gfCNCPoint1[11930] = {X 270.8909, Y 44.1700, Z -1.3333, A 0.000, B 0.000, C 0.000 }
gfCNCPoint1[11931] = {X 270.8910, Y 45.0000, Z -1.3333, A 0.000, B 0.000, C 0.000 }
gfCNCPoint1[11932] = {X 270.7867, Y 45.9257, Z -1.3333, A 0.000, B 0.000, C 0.000 }
gfCNCPoint1[11933] = {X 270.4791, Y 46.8050, Z -1.3333, A 0.000, B 0.000, C 0.000 }
gfCNCPoint1[11934] = {X 269.9835, Y 47.5937, Z -1.3333, A 0.000, B 0.000, C 0.000 }
gfCNCPoint1[11935] = {X 269.3247, Y 48.2524, Z -1.3333, A 0.000, B 0.000, C 0.000 }
gfCNCPoint1[11936] = {X 268.5360, Y 48.7480, Z -1.3333, A 0.000, B 0.000, C 0.000 }
gfCNCPoint1[11937] = {X 267.6567, Y 49.0557, Z -1.3333, A 0.000, B 0.000, C 0.000 }
gfCNCPoint1[11938] = {X 266.7310, Y 49.1600, Z -1.3333, A 0.000, B 0.000, C 0.000 }
gfCNCPoint1[11939] = {X 260.2876, Y 49.1600, Z -1.3333, A 0.000, B 0.000, C 0.000 }
gfCNCPoint1[11940] = {X 259.3664, Y 49.0567, Z -1.3333, A 0.000, B 0.000, C 0.000 }
gfCNCPoint1[11941] = {X 258.4910, Y 48.7520, Z -1.3333, A 0.000, B 0.000, C 0.000 }
gfCNCPoint1[11942] = {X 257.7047, Y 48.2611, Z -1.3333, A 0.000, B 0.000, C 0.000 }
gfCNCPoint1[11943] = {X 257.0467, Y 47.6082, Z -1.3333, A 0.000, B 0.000, C 0.000 }
gfCNCPoint1[11944] = {X 256.5496, Y 46.8258, Z -1.3333, A 0.000, B 0.000, C 0.000 }
gfCNCPoint1[11945] = {X 256.2381, Y 45.9527, Z -1.3333, A 0.000, B 0.000, C 0.000 }
gfCNCPoint1[11946] = {X 256.1277, Y 45.0324, Z -1.3333, A 0.000, B 0.000, C 0.000 }
gfCNCPoint1[11947] = {X 256.1280, Y 44.1516, Z -1.3333, A 0.000, B 0.000, C 0.000 }
gfCNCPoint1[11948] = {X 256.2385, Y 43.2545, Z -1.3333, A 0.000, B 0.000, C 0.000 }
gfCNCPoint1[11949] = {X 256.5401, Y 42.4026, Z -1.3333, A 0.000, B 0.000, C 0.000 }
gfCNCPoint1[11950] = {X 257.0187, Y 41.6358, Z -1.3333, A 0.000, B 0.000, C 0.000 }
gfCNCPoint1[11951] = {X 257.6515, Y 40.9906, Z -1.3333, A 0.000, B 0.000, C 0.000 }
gfCNCPoint1[11952] = {X 257.6515, Y 34.3138, Z -1.3333, A 0.000, B 0.000, C 0.000 }
gfCNCPoint1[11953] = {X 254.6687, Y 34.3138, Z -1.3333, A 0.000, B 0.000, C 0.000 }
gfCNCPoint1[11954] = {X 250.3098, Y 42.8058, Z -1.3333, A 0.000, B 0.000, C 0.000 }
gfCNCPoint1[11955] = {X 250.4891, Y 43.4795, Z -1.3333, A 0.000, B 0.000, C 0.000 }
gfCNCPoint1[11956] = {X 250.5534, Y 44.1736, Z -1.3333, A 0.000, B 0.000, C 0.000 }
gfCNCPoint1[11957] = {X 250.5536, Y 45.0000, Z -1.3333, A 0.000, B 0.000, C 0.000 }
gfCNCPoint1[11958] = {X 250.4493, Y 45.9257, Z -1.3333, A 0.000, B 0.000, C 0.000 }
gfCNCPoint1[11959] = {X 250.1416, Y 46.8050, Z -1.3333, A 0.000, B 0.000, C 0.000 }
gfCNCPoint1[11960] = {X 249.6460, Y 47.5937, Z -1.3333, A 0.000, B 0.000, C 0.000 }
gfCNCPoint1[11961] = {X 248.9873, Y 48.2524, Z -1.3333, A 0.000, B 0.000, C 0.000 }
gfCNCPoint1[11962] = {X 248.1985, Y 48.7480, Z -1.3333, A 0.000, B 0.000, C 0.000 }
gfCNCPoint1[11963] = {X 247.3192, Y 49.0557, Z -1.3333, A 0.000, B 0.000, C 0.000 }
gfCNCPoint1[11964] = {X 246.3936, Y 49.1600, Z -1.3333, A 0.000, B 0.000, C 0.000 }
gfCNCPoint1[11965] = {X 239.8075, Y 49.1600, Z -1.3333, A 0.000, B 0.000, C 0.000 }
gfCNCPoint1[11966] = {X 238.8818, Y 49.0557, Z -1.3333, A 0.000, B 0.000, C 0.000 }
gfCNCPoint1[11967] = {X 238.0026, Y 48.7480, Z -1.3333, A 0.000, B 0.000, C 0.000 }
gfCNCPoint1[11968] = {X 237.2138, Y 48.2524, Z -1.3333, A 0.000, B 0.000, C 0.000 }
gfCNCPoint1[11969] = {X 236.5551, Y 47.5937, Z -1.3333, A 0.000, B 0.000, C 0.000 }
gfCNCPoint1[11970] = {X 236.0595, Y 46.8050, Z -1.3333, A 0.000, B 0.000, C 0.000 }
gfCNCPoint1[11971] = {X 235.7518, Y 45.9257, Z -1.3333, A 0.000, B 0.000, C 0.000 }
gfCNCPoint1[11972] = {X 235.6475, Y 45.0000, Z -1.3333, A 0.000, B 0.000, C 0.000 }
gfCNCPoint1[11973] = {X 235.6479, Y 44.1516, Z -1.3333, A 0.000, B 0.000, C 0.000 }
gfCNCPoint1[11974] = {X 235.7441, Y 43.3174, Z -1.3333, A 0.000, B 0.000, C 0.000 }
gfCNCPoint1[11975] = {X 236.0059, Y 42.5195, Z -1.3333, A 0.000, B 0.000, C 0.000 }
gfCNCPoint1[11976] = {X 236.4226, Y 41.7905, Z -1.3333, A 0.000, B 0.000, C 0.000 }
gfCNCPoint1[11977] = {X 236.9772, Y 41.1600, Z -1.3333, A 0.000, B 0.000, C 0.000 }
gfCNCPoint1[11978] = {X 237.6471, Y 40.6537, Z -1.3333, A 0.000, B 0.000, C 0.000 }
gfCNCPoint1[11979] = {X 238.4051, Y 40.2923, Z -1.3333, A 0.000, B 0.000, C 0.000 }
gfCNCPoint1[11980] = {X 242.4925, Y 32.2917, Z -1.3333, A 0.000, B 0.000, C 0.000 }
gfCNCPoint1[11981] = {X 241.3086, Y 31.5171, Z -1.3333, A 0.000, B 0.000, C 0.000 }
gfCNCPoint1[11982] = {X 240.2323, Y 30.5990, Z -1.3333, A 0.000, B 0.000, C 0.000 }
gfCNCPoint1[11983] = {X 239.2808, Y 29.5520, Z -1.3333, A 0.000, B 0.000, C 0.000 }
gfCNCPoint1[11984] = {X 238.4695, Y 28.3930, Z -1.3333, A 0.000, B 0.000, C 0.000 }
gfCNCPoint1[11985] = {X 237.8114, Y 27.1407, Z -1.3333, A 0.000, B 0.000, C 0.000 }
gfCNCPoint1[11986] = {X 237.3171, Y 25.8152, Z -1.3333, A 0.000, B 0.000, C 0.000 }
gfCNCPoint1[11987] = {X 236.9012, Y 24.0214, Z -1.3333, A 0.000, B 0.000, C 0.000 }
gfCNCPoint1[11988] = {X 236.6893, Y 22.1924, Z -1.3333, A 0.000, B 0.000, C 0.000 }
gfCNCPoint1[11989] = {X 236.6841, Y 20.3511, Z -1.3333, A 0.000, B 0.000, C 0.000 }
gfCNCPoint1[11990] = {X 236.8856, Y 18.5208, Z -1.3333, A 0.000, B 0.000, C 0.000 }
gfCNCPoint1[11991] = {X 237.2914, Y 16.7248, Z -1.3333, A 0.000, B 0.000, C 0.000 }
gfCNCPoint1[11992] = {X 237.8539, Y 15.1704, Z -1.3333, A 0.000, B 0.000, C 0.000 }
gfCNCPoint1[11993] = {X 238.6302, Y 13.7110, Z -1.3333, A 0.000, B 0.000, C 0.000 }
gfCNCPoint1[11994] = {X 239.6047, Y 12.3757, Z -1.3333, A 0.000, B 0.000, C 0.000 }
gfCNCPoint1[11995] = {X 240.7578, Y 11.1913, Z -1.3333, A 0.000, B 0.000, C 0.000 }
gfCNCPoint1[11996] = {X 242.0665, Y 10.1815, Z -1.3333, A 0.000, B 0.000, C 0.000 }
gfCNCPoint1[11997] = {X 243.5046, Y 9.3664, Z -1.3333, A 0.000, B 0.000, C 0.000 }
gfCNCPoint1[11998] = {X 245.0434, Y 8.7624, Z -1.3333, A 0.000, B 0.000, C 0.000 }
gfCNCPoint1[11999] = {X 246.6520, Y 8.3817, Z -1.3333, A 0.000, B 0.000, C 0.000 }
gfCNCPoint1[12000] = {X 248.7352, Y 8.1119, Z -1.3333, A 0.000, B 0.000, C 0.000 }
gfCNCPoint1[12001] = {X 250.8343, Y 8.0319, Z -1.3333, A 0.000, B 0.000, C 0.000 }
gfCNCPoint1[12002] = {X 266.7621, Y 8.0319, Z -1.3333, A 0.000, B 0.000, C 0.000 }
gfCNCPoint1[12003] = {X 267.6817, Y 8.1424, Z -1.3333, A 0.000, B 0.000, C 0.000 }
gfCNCPoint1[12004] = {X 268.5541, Y 8.4535, Z -1.3333, A 0.000, B 0.000, C 0.000 }
gfCNCPoint1[12005] = {X 269.3361, Y 8.9499, Z -1.3333, A 0.000, B 0.000, C 0.000 }
gfCNCPoint1[12006] = {X 269.9891, Y 9.6069, Z -1.3333, A 0.000, B 0.000, C 0.000 }
gfCNCPoint1[12007] = {X 270.4805, Y 10.3920, Z -1.3333, A 0.000, B 0.000, C 0.000 }
gfCNCPoint1[12008] = {X 270.7862, Y 11.2663, Z -1.3333, A 0.000, B 0.000, C 0.000 }
gfCNCPoint1[12009] = {X 270.8910, Y 12.1866, Z -1.3333, A 0.000, B 0.000, C 0.000 }
gfCNCPoint1[12010] = {X 270.8908, Y 13.0208, Z -1.3333, A 0.000, B 0.000, C 0.000 }
gfCNCPoint1[12011] = {X 270.7823, Y 13.9231, Z -1.3333, A 0.000, B 0.000, C 0.000 }
gfCNCPoint1[12012] = {X 270.4804, Y 14.7802, Z -1.3333, A 0.000, B 0.000, C 0.000 }
gfCNCPoint1[12013] = {X 269.9996, Y 15.5514, Z -1.3333, A 0.000, B 0.000, C 0.000 }
gfCNCPoint1[12014] = {X 269.3628, Y 16.1997, Z -1.3333, A 0.000, B 0.000, C 0.000 }
gfCNCPoint1[12015] = {X 269.3627, Y 28.5937, Z -1.3333, A 0.000, B 0.000, C 0.000 }
gfCNCPoint1[12016] = {X 273.3627, Y 28.5937, Z -1.3333, A 0.000, B 0.000, C 0.000 }
gfCNCPoint1[12017] = {X 269.2827, Y 28.5937, Z -1.3333, A 0.000, B 0.000, C 0.000 }
gfCNCPoint1[12018] = {X 269.2826, Y 41.0279, Z -1.3333, A 0.000, B 0.000, C 0.000 }
gfCNCPoint1[12019] = {X 269.3835, Y 41.1087, Z -1.3333, A 0.000, B 0.000, C 0.000 }
gfCNCPoint1[12020] = {X 269.9800, Y 41.7409, Z -1.3333, A 0.000, B 0.000, C 0.000 }
gfCNCPoint1[12021] = {X 270.4290, Y 42.4851, Z -1.3333, A 0.000, B 0.000, C 0.000 }
gfCNCPoint1[12022] = {X 270.7102, Y 43.3075, Z -1.3333, A 0.000, B 0.000, C 0.000 }
gfCNCPoint1[12023] = {X 270.8109, Y 44.1708, Z -1.3333, A 0.000, B 0.000, C 0.000 }
gfCNCPoint1[12024] = {X 270.8110, Y 45.0000, Z -1.3333, A 0.000, B 0.000, C 0.000 }
gfCNCPoint1[12025] = {X 270.7087, Y 45.9079, Z -1.3333, A 0.000, B 0.000, C 0.000 }
gfCNCPoint1[12026] = {X 270.4070, Y 46.7702, Z -1.3333, A 0.000, B 0.000, C 0.000 }
gfCNCPoint1[12027] = {X 269.9209, Y 47.5438, Z -1.3333, A 0.000, B 0.000, C 0.000 }
gfCNCPoint1[12028] = {X 269.2749, Y 48.1899, Z -1.3333, A 0.000, B 0.000, C 0.000 }
gfCNCPoint1[12029] = {X 268.5013, Y 48.6760, Z -1.3333, A 0.000, B 0.000, C 0.000 }
gfCNCPoint1[12030] = {X 267.6389, Y 48.9777, Z -1.3333, A 0.000, B 0.000, C 0.000 }
gfCNCPoint1[12031] = {X 266.7310, Y 49.0800, Z -1.3333, A 0.000, B 0.000, C 0.000 }
gfCNCPoint1[12032] = {X 260.2876, Y 49.0800, Z -1.3333, A 0.000, B 0.000, C 0.000 }
gfCNCPoint1[12033] = {X 259.3841, Y 48.9787, Z -1.3333, A 0.000, B 0.000, C 0.000 }
gfCNCPoint1[12034] = {X 258.5255, Y 48.6799, Z -1.3333, A 0.000, B 0.000, C 0.000 }
gfCNCPoint1[12035] = {X 257.7544, Y 48.1983, Z -1.3333, A 0.000, B 0.000, C 0.000 }
gfCNCPoint1[12036] = {X 257.1090, Y 47.5580, Z -1.3333, A 0.000, B 0.000, C 0.000 }
gfCNCPoint1[12037] = {X 256.6215, Y 46.7907, Z -1.3333, A 0.000, B 0.000, C 0.000 }
gfCNCPoint1[12038] = {X 256.3160, Y 45.9344, Z -1.3333, A 0.000, B 0.000, C 0.000 }
gfCNCPoint1[12039] = {X 256.2077, Y 45.0318, Z -1.3333, A 0.000, B 0.000, C 0.000 }
gfCNCPoint1[12040] = {X 256.2080, Y 44.1527, Z -1.3333, A 0.000, B 0.000, C 0.000 }
gfCNCPoint1[12041] = {X 256.3185, Y 43.2637, Z -1.3333, A 0.000, B 0.000, C 0.000 }
gfCNCPoint1[12042] = {X 256.6204, Y 42.4203, Z -1.3333, A 0.000, B 0.000, C 0.000 }
gfCNCPoint1[12043] = {X 257.0991, Y 41.6631, Z -1.3333, A 0.000, B 0.000, C 0.000 }
gfCNCPoint1[12044] = {X 257.7315, Y 41.0287, Z -1.3333, A 0.000, B 0.000, C 0.000 }
gfCNCPoint1[12045] = {X 257.7315, Y 34.2338, Z -1.3333, A 0.000, B 0.000, C 0.000 }
gfCNCPoint1[12046] = {X 254.6199, Y 34.2338, Z -1.3333, A 0.000, B 0.000, C 0.000 }
gfCNCPoint1[12047] = {X 250.2227, Y 42.8003, Z -1.3333, A 0.000, B 0.000, C 0.000 }
gfCNCPoint1[12048] = {X 250.4073, Y 43.4765, Z -1.3333, A 0.000, B 0.000, C 0.000 }
gfCNCPoint1[12049] = {X 250.4734, Y 44.1743, Z -1.3333, A 0.000, B 0.000, C 0.000 }
gfCNCPoint1[12050] = {X 250.4736, Y 45.0000, Z -1.3333, A 0.000, B 0.000, C 0.000 }
gfCNCPoint1[12051] = {X 250.3713, Y 45.9079, Z -1.3333, A 0.000, B 0.000, C 0.000 }
gfCNCPoint1[12052] = {X 250.0695, Y 46.7702, Z -1.3333, A 0.000, B 0.000, C 0.000 }
gfCNCPoint1[12053] = {X 249.5834, Y 47.5438, Z -1.3333, A 0.000, B 0.000, C 0.000 }
gfCNCPoint1[12054] = {X 248.9374, Y 48.1899, Z -1.3333, A 0.000, B 0.000, C 0.000 }
gfCNCPoint1[12055] = {X 248.1638, Y 48.6760, Z -1.3333, A 0.000, B 0.000, C 0.000 }
gfCNCPoint1[12056] = {X 247.3014, Y 48.9777, Z -1.3333, A 0.000, B 0.000, C 0.000 }
gfCNCPoint1[12057] = {X 246.3936, Y 49.0800, Z -1.3333, A 0.000, B 0.000, C 0.000 }
gfCNCPoint1[12058] = {X 239.8075, Y 49.0800, Z -1.3333, A 0.000, B 0.000, C 0.000 }
gfCNCPoint1[12059] = {X 238.8996, Y 48.9777, Z -1.3333, A 0.000, B 0.000, C 0.000 }
gfCNCPoint1[12060] = {X 238.0373, Y 48.6760, Z -1.3333, A 0.000, B 0.000, C 0.000 }
gfCNCPoint1[12061] = {X 237.2637, Y 48.1899, Z -1.3333, A 0.000, B 0.000, C 0.000 }
gfCNCPoint1[12062] = {X 236.6176, Y 47.5438, Z -1.3333, A 0.000, B 0.000, C 0.000 }
gfCNCPoint1[12063] = {X 236.1315, Y 46.7702, Z -1.3333, A 0.000, B 0.000, C 0.000 }
gfCNCPoint1[12064] = {X 235.8298, Y 45.9079, Z -1.3333, A 0.000, B 0.000, C 0.000 }
gfCNCPoint1[12065] = {X 235.7275, Y 45.0000, Z -1.3333, A 0.000, B 0.000, C 0.000 }
gfCNCPoint1[12066] = {X 235.7279, Y 44.1527, Z -1.3333, A 0.000, B 0.000, C 0.000 }
gfCNCPoint1[12067] = {X 235.8234, Y 43.3294, Z -1.3333, A 0.000, B 0.000, C 0.000 }
gfCNCPoint1[12068] = {X 236.0833, Y 42.5424, Z -1.3333, A 0.000, B 0.000, C 0.000 }
gfCNCPoint1[12069] = {X 236.4969, Y 41.8242, Z -1.3333, A 0.000, B 0.000, C 0.000 }
gfCNCPoint1[12070] = {X 237.0471, Y 41.2044, Z -1.3333, A 0.000, B 0.000, C 0.000 }
gfCNCPoint1[12071] = {X 237.7112, Y 40.7085, Z -1.3333, A 0.000, B 0.000, C 0.000 }
gfCNCPoint1[12072] = {X 238.4618, Y 40.3571, Z -1.3333, A 0.000, B 0.000, C 0.000 }
gfCNCPoint1[12073] = {X 242.5987, Y 32.2596, Z -1.3333, A 0.000, B 0.000, C 0.000 }
gfCNCPoint1[12074] = {X 241.4078, Y 31.4912, Z -1.3333, A 0.000, B 0.000, C 0.000 }
gfCNCPoint1[12075] = {X 240.3247, Y 30.5770, Z -1.3333, A 0.000, B 0.000, C 0.000 }
